REGION Network 5
   RUNG wire#powerrail
      "S2_Interlocks_DB"(Vessel_Rad_Level := "S2_General_Setup".Vessel_Rad_Level, Vessel_Rad_High_Alarm := "S2_General_Setup".Vessel_Alarm_Level, Pump_Rad_Level := "S2_General_Setup".Pump_Rad_Level, Pump_Rad_High_Alarm := "S2_General_Setup".Pump_Alarm_Level, Estop1 := "Estop1_PB_Active", Estop2 := "Estop2_PB_Active", Safety_Relay_Trip := "Safety_Relay_Trip", Safety_Lock_Engaged := "Safety_Lock2_Engaged", Manual_Mode := "S2_General_Setup".Manual_Mode, Rad_Lock_Bypass := "S2_General_Setup".Rad_Lock_Bypass, Process_Complete := "S2_General_Setup".Auto_Process_Complete, Water_Supply_Interlock := "S2_General_Setup".Water_Supply_Interlock, UM_Container_Interlock := "Setup_Data".Waste_Container_Interlock, UM_Container_HH_Interlock := "UM_HI_Level_SW", Buzzer_Reset := "Setup_Data".Buzzer_Reset, Rad_Lock := "S2_General_Setup".Rad_Lock, Estop_Active := "Setup_Data".Estop_Active, Level_Interlock := "S2_General_Setup".Level_Interlock, Pump_Permisive => "Pmp2_Permissive")
   END_RUNG
   // the same network as SCL:
   "S2_Interlocks_DB"(Vessel_Rad_Level := "S2_General_Setup".Vessel_Rad_Level,   // "Interlocks"
                      Vessel_Rad_High_Alarm := "S2_General_Setup".Vessel_Alarm_Level,
                      Pump_Rad_Level := "S2_General_Setup".Pump_Rad_Level,
                      Pump_Rad_High_Alarm := "S2_General_Setup".Pump_Alarm_Level,
                      Estop1 := "Estop1_PB_Active",
                      Estop2 := "Estop2_PB_Active",
                      Safety_Relay_Trip := "Safety_Relay_Trip",
                      Safety_Lock_Engaged := "Safety_Lock2_Engaged",
                      Manual_Mode := "S2_General_Setup".Manual_Mode,
                      Rad_Lock_Bypass := "S2_General_Setup".Rad_Lock_Bypass,
                      Process_Complete := "S2_General_Setup".Auto_Process_Complete,
                      Water_Supply_Interlock := "S2_General_Setup".Water_Supply_Interlock,
                      UM_Container_Interlock := "Setup_Data".Waste_Container_Interlock,
                      UM_Container_HH_Interlock := "UM_HI_Level_SW",
                      Buzzer_Reset := "Setup_Data".Buzzer_Reset,
                      Rad_Lock := "S2_General_Setup".Rad_Lock,
                      Estop_Active := "Setup_Data".Estop_Active,
                      Level_Interlock := "S2_General_Setup".Level_Interlock,
                      Pump_Permisive => "Pmp2_Permissive");
END_REGION

REGION Network 6
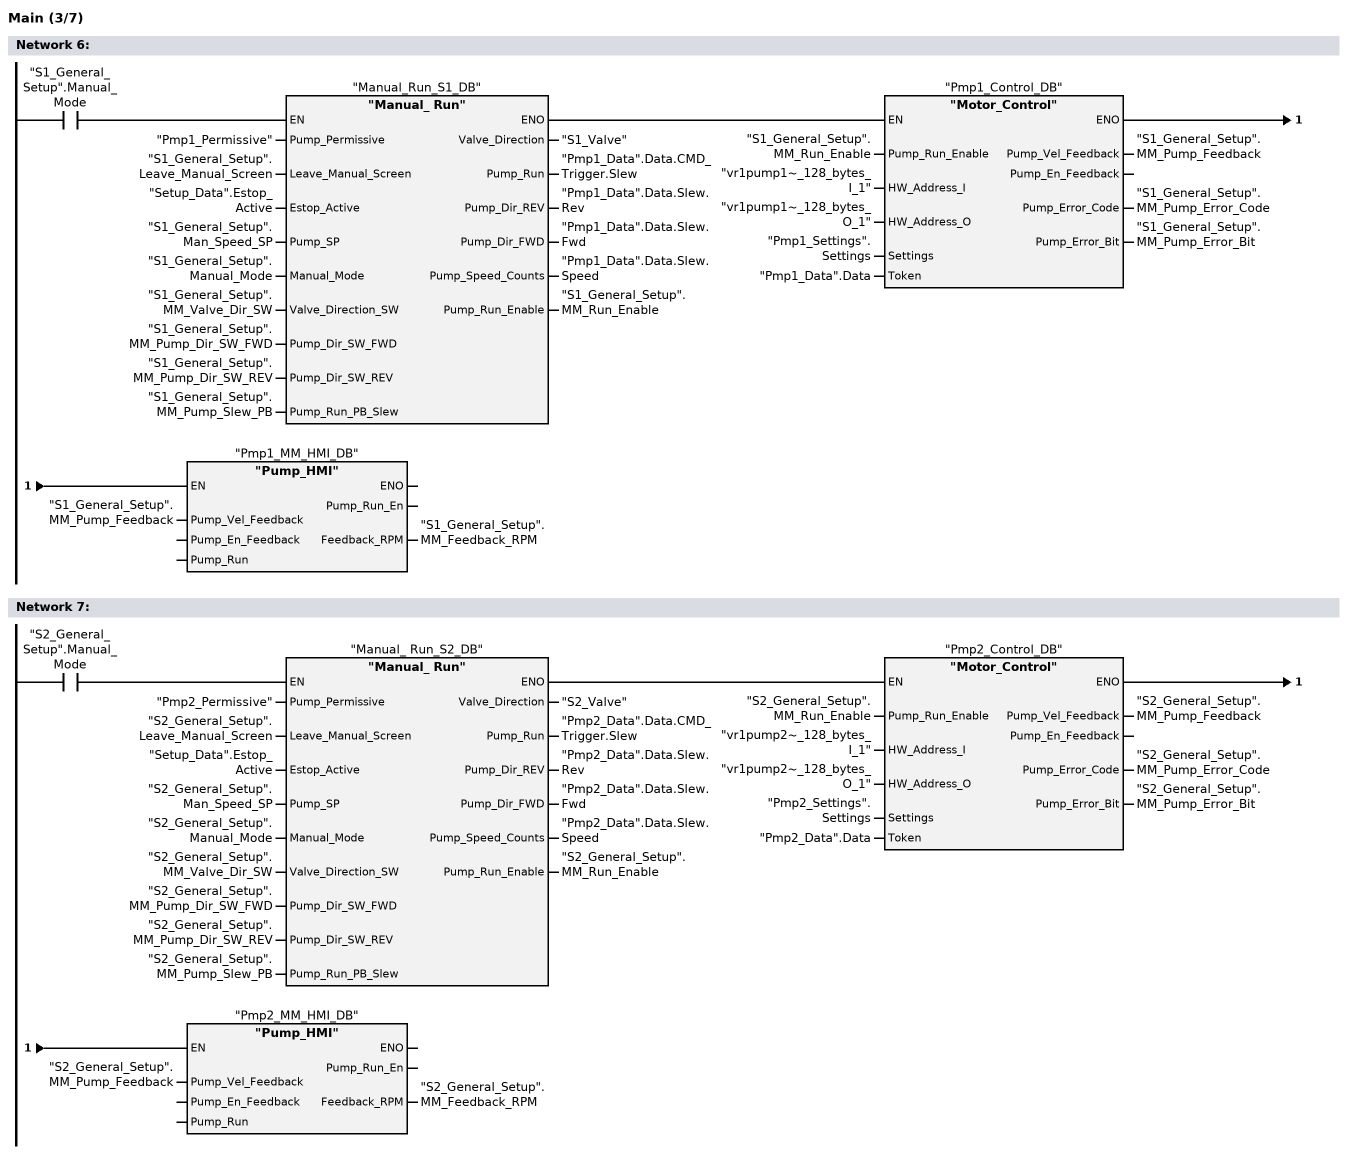
   RUNG wire#powerrail
      Contact( "S1_General_Setup".Manual_Mode )
      "Manual_Run_S1_DB"(Pump_Permissive := "Pmp1_Permissive", Leave_Manual_Screen := "S1_General_Setup".Leave_Manual_Screen, Estop_Active := "Setup_Data".Estop_Active, Pump_SP := "S1_General_Setup".Man_Speed_SP, Manual_Mode := "S1_General_Setup".Manual_Mode, Valve_Direction_SW := "S1_General_Setup".MM_Valve_Dir_SW, Pump_Dir_SW_FWD := "S1_General_Setup".MM_Pump_Dir_SW_FWD, Pump_Dir_SW_REV := "S1_General_Setup".MM_Pump_Dir_SW_REV, Pump_Run_PB_Slew := "S1_General_Setup".MM_Pump_Slew_PB, Valve_Direction => "S1_Valve", Pump_Run => "Pmp1_Data".Data.CMD_Trigger.Slew, Pump_Dir_REV => "Pmp1_Data".Data.Slew.Rev, Pump_Dir_FWD => "Pmp1_Data".Data.Slew.Fwd, Pump_Speed_Counts => "Pmp1_Data".Data.Slew.Speed, Pump_Run_Enable => "S1_General_Setup".MM_Run_Enable)
      "Pmp1_Control_DB"(Pump_Run_Enable := "S1_General_Setup".MM_Run_Enable, HW_Address_I := "vr1pump1~_128_bytes_I_1", HW_Address_O := "vr1pump1~_128_bytes_O_1", Settings := "Pmp1_Settings".Settings, Token := "Pmp1_Data".Data, Pump_Vel_Feedback => "S1_General_Setup".MM_Pump_Feedback, Pump_En_Feedback =>, Pump_Error_Code => "S1_General_Setup".MM_Pump_Error_Code, Pump_Error_Bit => "S1_General_Setup".MM_Pump_Error_Bit)
      "Pmp1_MM_HMI_DB"(Pump_Vel_Feedback := "S1_General_Setup".MM_Pump_Feedback, Pump_En_Feedback :=, Pump_Run :=, Pump_Run_En =>, Feedback_RPM => "S1_General_Setup".MM_Feedback_RPM)
   END_RUNG
   // the same network as SCL:
   "Manual_Run_S1_DB"(EN := "S1_General_Setup".Manual_Mode,   // "Manual_ Run"
                      Pump_Permissive := "Pmp1_Permissive",
                      Leave_Manual_Screen := "S1_General_Setup".Leave_Manual_Screen,
                      Estop_Active := "Setup_Data".Estop_Active,
                      Pump_SP := "S1_General_Setup".Man_Speed_SP,
                      Manual_Mode := "S1_General_Setup".Manual_Mode,
                      Valve_Direction_SW := "S1_General_Setup".MM_Valve_Dir_SW,
                      Pump_Dir_SW_FWD := "S1_General_Setup".MM_Pump_Dir_SW_FWD,
                      Pump_Dir_SW_REV := "S1_General_Setup".MM_Pump_Dir_SW_REV,
                      Pump_Run_PB_Slew := "S1_General_Setup".MM_Pump_Slew_PB,
                      Valve_Direction => "S1_Valve",
                      Pump_Run => "Pmp1_Data".Data.CMD_Trigger.Slew,
                      Pump_Dir_REV => "Pmp1_Data".Data.Slew.Rev,
                      Pump_Dir_FWD => "Pmp1_Data".Data.Slew.Fwd,
                      Pump_Speed_Counts => "Pmp1_Data".Data.Slew.Speed,
                      Pump_Run_Enable => "S1_General_Setup".MM_Run_Enable,
                      ENO => #_w1);
   "Pmp1_Control_DB"(EN := #_w1,   // "Motor_Control"
                     Pump_Run_Enable := "S1_General_Setup".MM_Run_Enable,
                     HW_Address_I := "vr1pump1~_128_bytes_I_1",
                     HW_Address_O := "vr1pump1~_128_bytes_O_1",
                     Settings := "Pmp1_Settings".Settings,
                     Token := "Pmp1_Data".Data,
                     Pump_Vel_Feedback => "S1_General_Setup".MM_Pump_Feedback,
                     Pump_Error_Code => "S1_General_Setup".MM_Pump_Error_Code,
                     Pump_Error_Bit => "S1_General_Setup".MM_Pump_Error_Bit,
                     ENO => #_w2);
   IF #_w2 THEN
       "Pmp1_MM_HMI_DB"(Pump_Vel_Feedback := "S1_General_Setup".MM_Pump_Feedback,   // "Pump_HMI"
                        Feedback_RPM => "S1_General_Setup".MM_Feedback_RPM);
   END_IF;
END_REGION

REGION Network 7
   RUNG wire#powerrail
      Contact( "S2_General_Setup".Manual_Mode )
      "Manual_ Run_S2_DB"(Pump_Permissive := "Pmp2_Permissive", Leave_Manual_Screen := "S2_General_Setup".Leave_Manual_Screen, Estop_Active := "Setup_Data".Estop_Active, Pump_SP := "S2_General_Setup".Man_Speed_SP, Manual_Mode := "S2_General_Setup".Manual_Mode, Valve_Direction_SW := "S2_General_Setup".MM_Valve_Dir_SW, Pump_Dir_SW_FWD := "S2_General_Setup".MM_Pump_Dir_SW_FWD, Pump_Dir_SW_REV := "S2_General_Setup".MM_Pump_Dir_SW_REV, Pump_Run_PB_Slew := "S2_General_Setup".MM_Pump_Slew_PB, Valve_Direction => "S2_Valve", Pump_Run => "Pmp2_Data".Data.CMD_Trigger.Slew, Pump_Dir_REV => "Pmp2_Data".Data.Slew.Rev, Pump_Dir_FWD => "Pmp2_Data".Data.Slew.Fwd, Pump_Speed_Counts => "Pmp2_Data".Data.Slew.Speed, Pump_Run_Enable => "S2_General_Setup".MM_Run_Enable)
      "Pmp2_Control_DB"(Pump_Run_Enable := "S2_General_Setup".MM_Run_Enable, HW_Address_I := "vr1pump2~_128_bytes_I_1", HW_Address_O := "vr1pump2~_128_bytes_O_1", Settings := "Pmp2_Settings".Settings, Token := "Pmp2_Data".Data, Pump_Vel_Feedback => "S2_General_Setup".MM_Pump_Feedback, Pump_En_Feedback =>, Pump_Error_Code => "S2_General_Setup".MM_Pump_Error_Code, Pump_Error_Bit => "S2_General_Setup".MM_Pump_Error_Bit)
      "Pmp2_MM_HMI_DB"(Pump_Vel_Feedback := "S2_General_Setup".MM_Pump_Feedback, Pump_En_Feedback :=, Pump_Run :=, Pump_Run_En =>, Feedback_RPM => "S2_General_Setup".MM_Feedback_RPM)
   END_RUNG
   // the same network as SCL:
   "Manual_ Run_S2_DB"(EN := "S2_General_Setup".Manual_Mode,   // "Manual_ Run"
                       Pump_Permissive := "Pmp2_Permissive",
                       Leave_Manual_Screen := "S2_General_Setup".Leave_Manual_Screen,
                       Estop_Active := "Setup_Data".Estop_Active,
                       Pump_SP := "S2_General_Setup".Man_Speed_SP,
                       Manual_Mode := "S2_General_Setup".Manual_Mode,
                       Valve_Direction_SW := "S2_General_Setup".MM_Valve_Dir_SW,
                       Pump_Dir_SW_FWD := "S2_General_Setup".MM_Pump_Dir_SW_FWD,
                       Pump_Dir_SW_REV := "S2_General_Setup".MM_Pump_Dir_SW_REV,
                       Pump_Run_PB_Slew := "S2_General_Setup".MM_Pump_Slew_PB,
                       Valve_Direction => "S2_Valve",
                       Pump_Run => "Pmp2_Data".Data.CMD_Trigger.Slew,
                       Pump_Dir_REV => "Pmp2_Data".Data.Slew.Rev,
                       Pump_Dir_FWD => "Pmp2_Data".Data.Slew.Fwd,
                       Pump_Speed_Counts => "Pmp2_Data".Data.Slew.Speed,
                       Pump_Run_Enable => "S2_General_Setup".MM_Run_Enable,
                       ENO => #_w1);
   "Pmp2_Control_DB"(EN := #_w1,   // "Motor_Control"
                     Pump_Run_Enable := "S2_General_Setup".MM_Run_Enable,
                     HW_Address_I := "vr1pump2~_128_bytes_I_1",
                     HW_Address_O := "vr1pump2~_128_bytes_O_1",
                     Settings := "Pmp2_Settings".Settings,
                     Token := "Pmp2_Data".Data,
                     Pump_Vel_Feedback => "S2_General_Setup".MM_Pump_Feedback,
                     Pump_Error_Code => "S2_General_Setup".MM_Pump_Error_Code,
                     Pump_Error_Bit => "S2_General_Setup".MM_Pump_Error_Bit,
                     ENO => #_w2);
   IF #_w2 THEN
       "Pmp2_MM_HMI_DB"(Pump_Vel_Feedback := "S2_General_Setup".MM_Pump_Feedback,   // "Pump_HMI"
                        Feedback_RPM => "S2_General_Setup".MM_Feedback_RPM);
   END_IF;
END_REGION

REGION Network 8
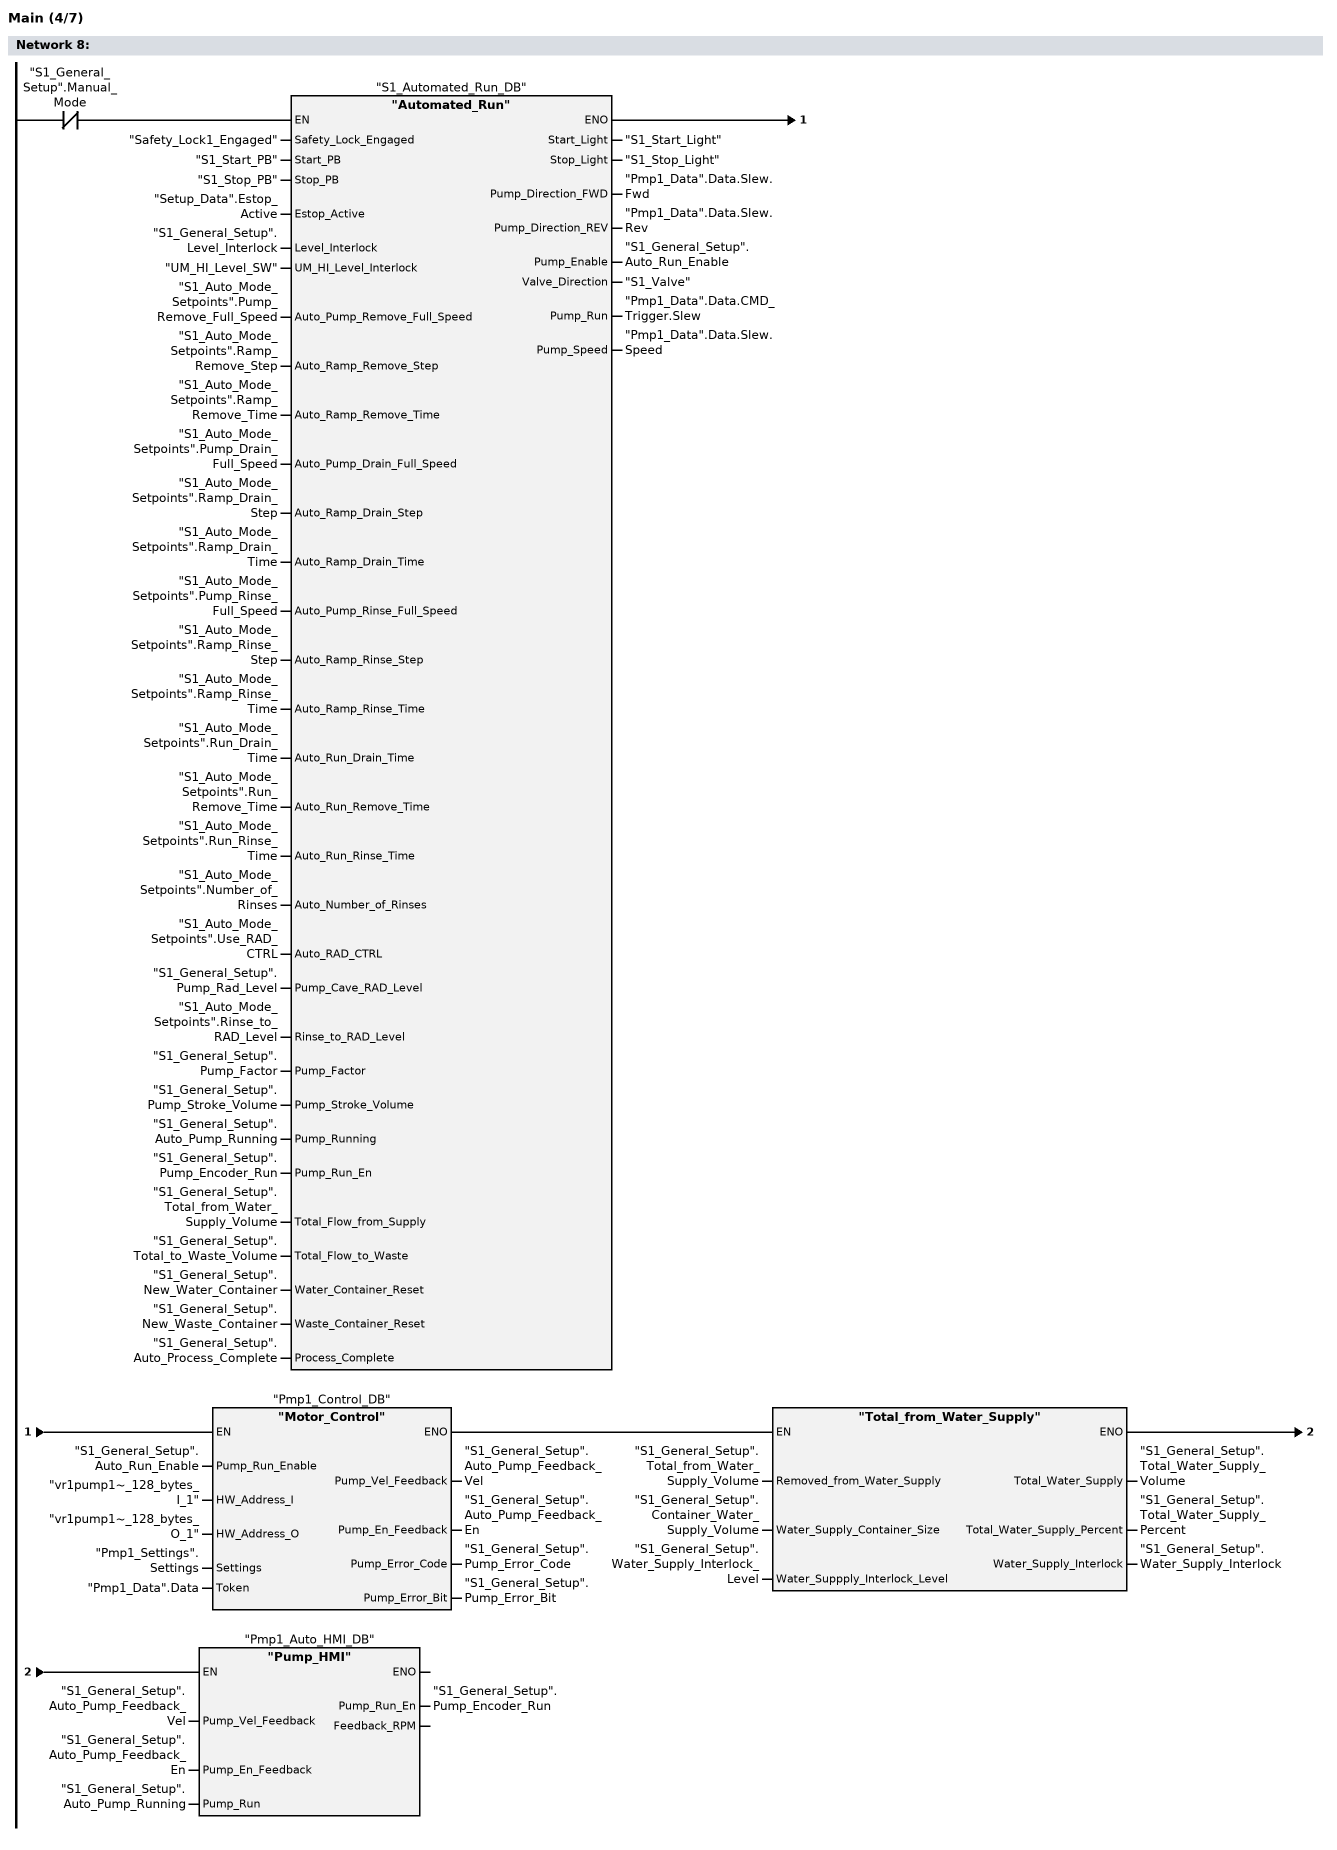
   RUNG wire#powerrail
      I_Contact( "S1_General_Setup".Manual_Mode )
      "S1_Automated_Run_DB"(Safety_Lock_Engaged := "Safety_Lock1_Engaged", Start_PB := "S1_Start_PB", Stop_PB := "S1_Stop_PB", Estop_Active := "Setup_Data".Estop_Active, Level_Interlock := "S1_General_Setup".Level_Interlock, UM_HI_Level_Interlock := "UM_HI_Level_SW", Auto_Pump_Remove_Full_Speed := "S1_Auto_Mode_Setpoints".Pump_Remove_Full_Speed, Auto_Ramp_Remove_Step := "S1_Auto_Mode_Setpoints".Ramp_Remove_Step, Auto_Ramp_Remove_Time := "S1_Auto_Mode_Setpoints".Ramp_Remove_Time, Auto_Pump_Drain_Full_Speed := "S1_Auto_Mode_Setpoints".Pump_Drain_Full_Speed, Auto_Ramp_Drain_Step := "S1_Auto_Mode_Setpoints".Ramp_Drain_Step, Auto_Ramp_Drain_Time := "S1_Auto_Mode_Setpoints".Ramp_Drain_Time, Auto_Pump_Rinse_Full_Speed := "S1_Auto_Mode_Setpoints".Pump_Rinse_Full_Speed, Auto_Ramp_Rinse_Step := "S1_Auto_Mode_Setpoints".Ramp_Rinse_Step, Auto_Ramp_Rinse_Time := "S1_Auto_Mode_Setpoints".Ramp_Rinse_Time, Auto_Run_Drain_Time := "S1_Auto_Mode_Setpoints".Run_Drain_Time, Auto_Run_Remove_Time := "S1_Auto_Mode_Setpoints".Run_Remove_Time, Auto_Run_Rinse_Time := "S1_Auto_Mode_Setpoints".Run_Rinse_Time, Auto_Number_of_Rinses := "S1_Auto_Mode_Setpoints".Number_of_Rinses, Auto_RAD_CTRL := "S1_Auto_Mode_Setpoints".Use_RAD_CTRL, Pump_Cave_RAD_Level := "S1_General_Setup".Pump_Rad_Level, Rinse_to_RAD_Level := "S1_Auto_Mode_Setpoints".Rinse_to_RAD_Level, Pump_Factor := "S1_General_Setup".Pump_Factor, Pump_Stroke_Volume := "S1_General_Setup".Pump_Stroke_Volume, Pump_Running := "S1_General_Setup".Auto_Pump_Running, Pump_Run_En := "S1_General_Setup".Pump_Encoder_Run, Total_Flow_from_Supply := "S1_General_Setup".Total_from_Water_Supply_Volume, Total_Flow_to_Waste := "S1_General_Setup".Total_to_Waste_Volume, Water_Container_Reset := "S1_General_Setup".New_Water_Container, Waste_Container_Reset := "S1_General_Setup".New_Waste_Container, Process_Complete := "S1_General_Setup".Auto_Process_Complete, Start_Light => "S1_Start_Light", Stop_Light => "S1_Stop_Light", Pump_Direction_FWD => "Pmp1_Data".Data.Slew.Fwd, Pump_Direction_REV => "Pmp1_Data".Data.Slew.Rev, Pump_Enable => "S1_General_Setup".Auto_Run_Enable, Valve_Direction => "S1_Valve", Pump_Run => "Pmp1_Data".Data.CMD_Trigger.Slew, Pump_Speed => "Pmp1_Data".Data.Slew.Speed)
      "Pmp1_Control_DB"(Pump_Run_Enable := "S1_General_Setup".Auto_Run_Enable, HW_Address_I := "vr1pump1~_128_bytes_I_1", HW_Address_O := "vr1pump1~_128_bytes_O_1", Settings := "Pmp1_Settings".Settings, Token := "Pmp1_Data".Data, Pump_Vel_Feedback => "S1_General_Setup".Auto_Pump_Feedback_Vel, Pump_En_Feedback => "S1_General_Setup".Auto_Pump_Feedback_En, Pump_Error_Code => "S1_General_Setup".Pump_Error_Code, Pump_Error_Bit => "S1_General_Setup".Pump_Error_Bit)
      "Total_from_Water_Supply"(Removed_from_Water_Supply := "S1_General_Setup".Total_from_Water_Supply_Volume, Water_Supply_Container_Size := "S1_General_Setup".Container_Water_Supply_Volume, Water_Suppply_Interlock_Level := "S1_General_Setup".Water_Supply_Interlock_Level, Total_Water_Supply => "S1_General_Setup".Total_Water_Supply_Volume, Total_Water_Supply_Percent => "S1_General_Setup".Total_Water_Supply_Percent, Water_Supply_Interlock => "S1_General_Setup".Water_Supply_Interlock)
      "Pmp1_Auto_HMI_DB"(Pump_Vel_Feedback := "S1_General_Setup".Auto_Pump_Feedback_Vel, Pump_En_Feedback := "S1_General_Setup".Auto_Pump_Feedback_En, Pump_Run := "S1_General_Setup".Auto_Pump_Running, Pump_Run_En => "S1_General_Setup".Pump_Encoder_Run, Feedback_RPM =>)
   END_RUNG
   // the same network as SCL:
   "S1_Automated_Run_DB"(EN := NOT "S1_General_Setup".Manual_Mode,   // "Automated_Run"
                         Safety_Lock_Engaged := "Safety_Lock1_Engaged",
                         Start_PB := "S1_Start_PB",
                         Stop_PB := "S1_Stop_PB",
                         Estop_Active := "Setup_Data".Estop_Active,
                         Level_Interlock := "S1_General_Setup".Level_Interlock,
                         UM_HI_Level_Interlock := "UM_HI_Level_SW",
                         Auto_Pump_Remove_Full_Speed := "S1_Auto_Mode_Setpoints".Pump_Remove_Full_Speed,
                         Auto_Ramp_Remove_Step := "S1_Auto_Mode_Setpoints".Ramp_Remove_Step,
                         Auto_Ramp_Remove_Time := "S1_Auto_Mode_Setpoints".Ramp_Remove_Time,
                         Auto_Pump_Drain_Full_Speed := "S1_Auto_Mode_Setpoints".Pump_Drain_Full_Speed,
                         Auto_Ramp_Drain_Step := "S1_Auto_Mode_Setpoints".Ramp_Drain_Step,
                         Auto_Ramp_Drain_Time := "S1_Auto_Mode_Setpoints".Ramp_Drain_Time,
                         Auto_Pump_Rinse_Full_Speed := "S1_Auto_Mode_Setpoints".Pump_Rinse_Full_Speed,
                         Auto_Ramp_Rinse_Step := "S1_Auto_Mode_Setpoints".Ramp_Rinse_Step,
                         Auto_Ramp_Rinse_Time := "S1_Auto_Mode_Setpoints".Ramp_Rinse_Time,
                         Auto_Run_Drain_Time := "S1_Auto_Mode_Setpoints".Run_Drain_Time,
                         Auto_Run_Remove_Time := "S1_Auto_Mode_Setpoints".Run_Remove_Time,
                         Auto_Run_Rinse_Time := "S1_Auto_Mode_Setpoints".Run_Rinse_Time,
                         Auto_Number_of_Rinses := "S1_Auto_Mode_Setpoints".Number_of_Rinses,
                         Auto_RAD_CTRL := "S1_Auto_Mode_Setpoints".Use_RAD_CTRL,
                         Pump_Cave_RAD_Level := "S1_General_Setup".Pump_Rad_Level,
                         Rinse_to_RAD_Level := "S1_Auto_Mode_Setpoints".Rinse_to_RAD_Level,
                         Pump_Factor := "S1_General_Setup".Pump_Factor,
                         Pump_Stroke_Volume := "S1_General_Setup".Pump_Stroke_Volume,
                         Pump_Running := "S1_General_Setup".Auto_Pump_Running,
                         Pump_Run_En := "S1_General_Setup".Pump_Encoder_Run,
                         Total_Flow_from_Supply := "S1_General_Setup".Total_from_Water_Supply_Volume,
                         Total_Flow_to_Waste := "S1_General_Setup".Total_to_Waste_Volume,
                         Water_Container_Reset := "S1_General_Setup".New_Water_Container,
                         Waste_Container_Reset := "S1_General_Setup".New_Waste_Container,
                         Process_Complete := "S1_General_Setup".Auto_Process_Complete,
                         Start_Light => "S1_Start_Light",
                         Stop_Light => "S1_Stop_Light",
                         Pump_Direction_FWD => "Pmp1_Data".Data.Slew.Fwd,
                         Pump_Direction_REV => "Pmp1_Data".Data.Slew.Rev,
                         Pump_Enable => "S1_General_Setup".Auto_Run_Enable,
                         Valve_Direction => "S1_Valve",
                         Pump_Run => "Pmp1_Data".Data.CMD_Trigger.Slew,
                         Pump_Speed => "Pmp1_Data".Data.Slew.Speed,
                         ENO => #_w1);
   "Pmp1_Control_DB"(EN := #_w1,   // "Motor_Control"
                     Pump_Run_Enable := "S1_General_Setup".Auto_Run_Enable,
                     HW_Address_I := "vr1pump1~_128_bytes_I_1",
                     HW_Address_O := "vr1pump1~_128_bytes_O_1",
                     Settings := "Pmp1_Settings".Settings,
                     Token := "Pmp1_Data".Data,
                     Pump_Vel_Feedback => "S1_General_Setup".Auto_Pump_Feedback_Vel,
                     Pump_En_Feedback => "S1_General_Setup".Auto_Pump_Feedback_En,
                     Pump_Error_Code => "S1_General_Setup".Pump_Error_Code,
                     Pump_Error_Bit => "S1_General_Setup".Pump_Error_Bit,
                     ENO => #_w2);
   "Total_from_Water_Supply"(EN := #_w2,
                           Removed_from_Water_Supply := "S1_General_Setup".Total_from_Water_Supply_Volume,
                           Water_Supply_Container_Size := "S1_General_Setup".Container_Water_Supply_Volume,
                           Water_Suppply_Interlock_Level := "S1_General_Setup".Water_Supply_Interlock_Level,
                           Total_Water_Supply => "S1_General_Setup".Total_Water_Supply_Volume,
                           Total_Water_Supply_Percent => "S1_General_Setup".Total_Water_Supply_Percent,
                           Water_Supply_Interlock => "S1_General_Setup".Water_Supply_Interlock,
                           ENO => #_w3);
   IF #_w3 THEN
       "Pmp1_Auto_HMI_DB"(Pump_Vel_Feedback := "S1_General_Setup".Auto_Pump_Feedback_Vel,   // "Pump_HMI"
                          Pump_En_Feedback := "S1_General_Setup".Auto_Pump_Feedback_En,
                          Pump_Run := "S1_General_Setup".Auto_Pump_Running,
                          Pump_Run_En => "S1_General_Setup".Pump_Encoder_Run);
   END_IF;
END_REGION

REGION Network 9
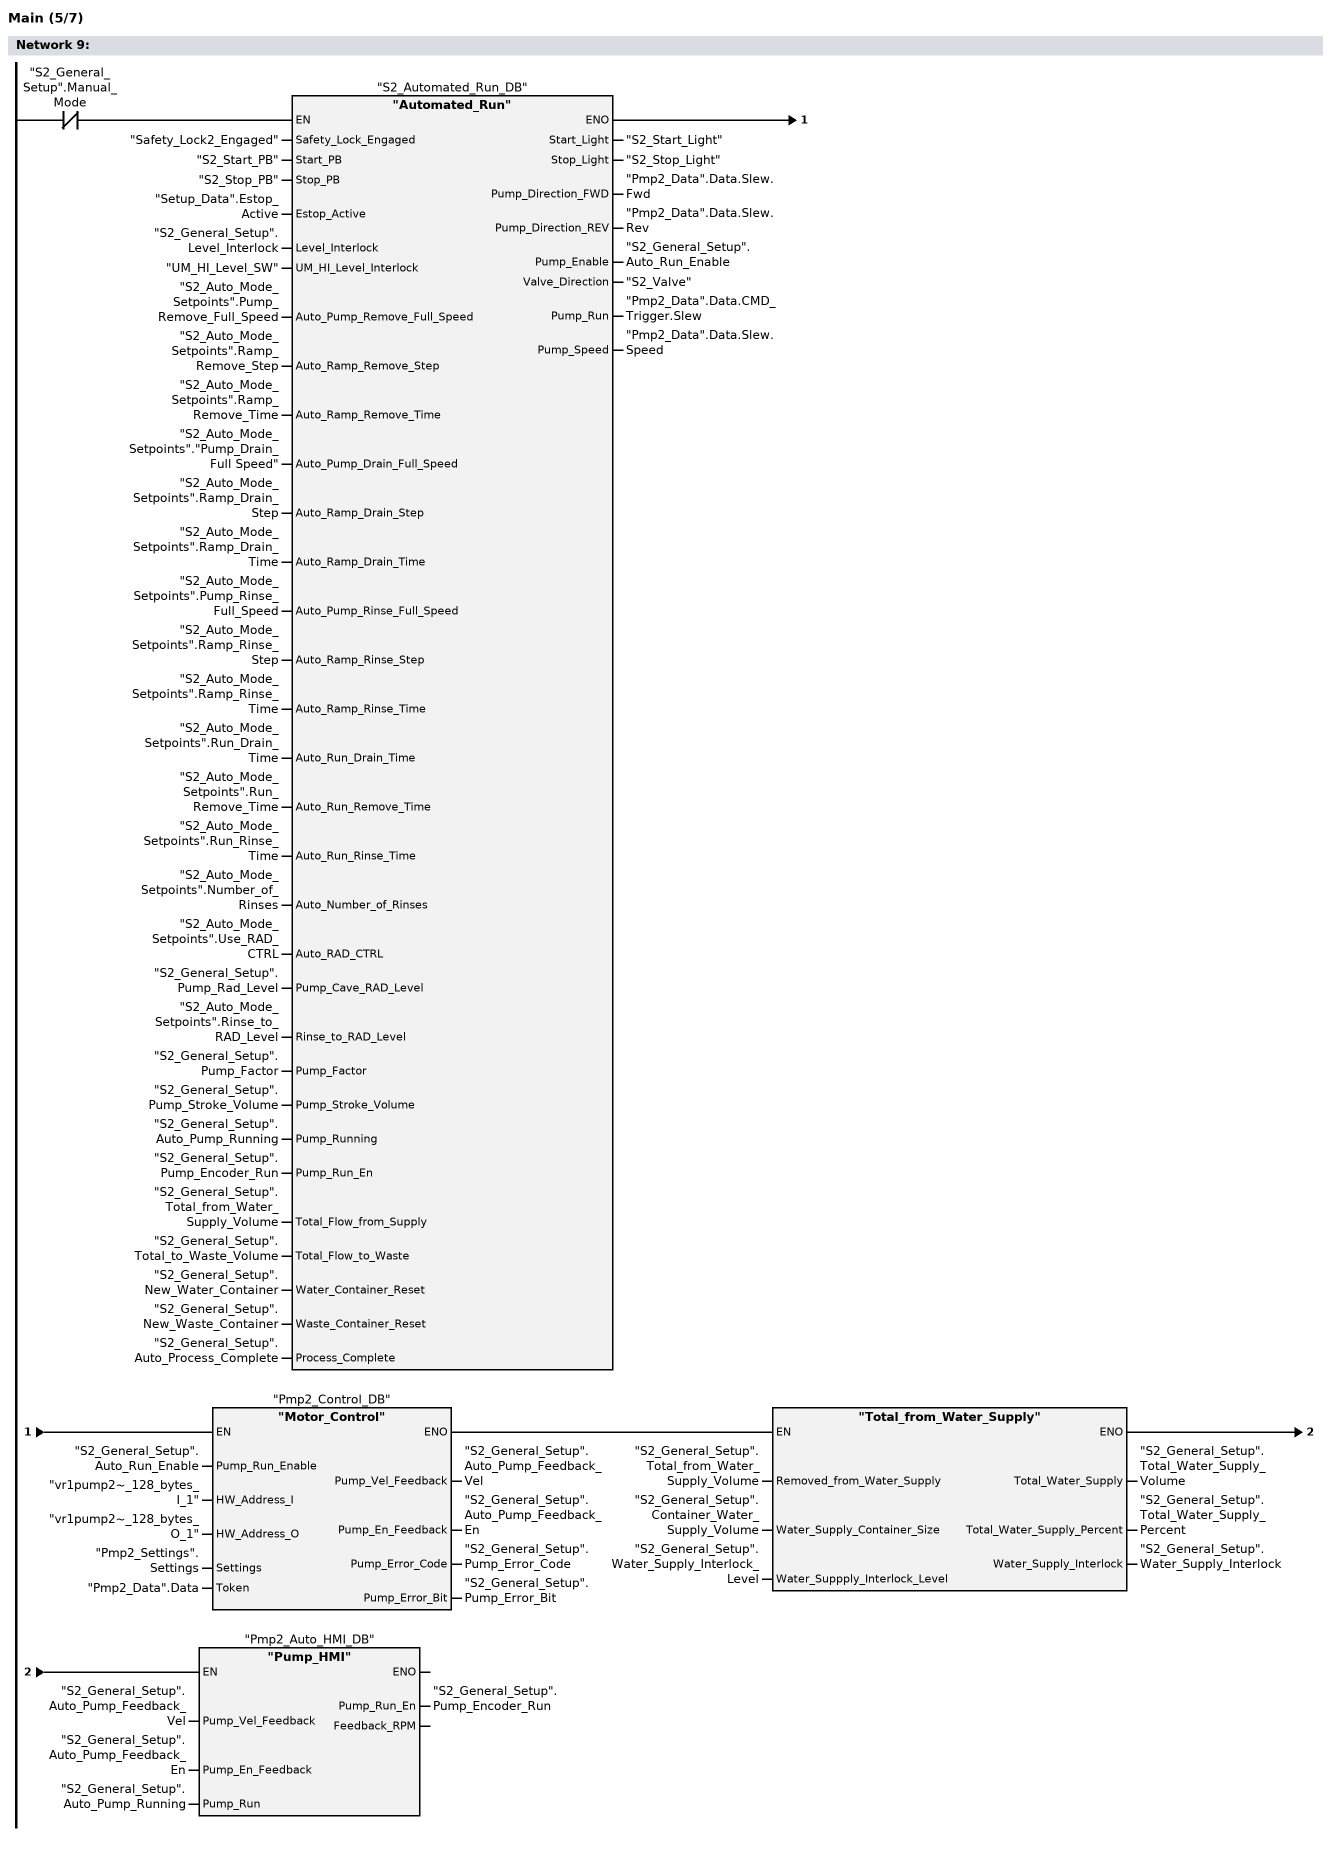
   RUNG wire#powerrail
      I_Contact( "S2_General_Setup".Manual_Mode )
      "S2_Automated_Run_DB"(Safety_Lock_Engaged := "Safety_Lock2_Engaged", Start_PB := "S2_Start_PB", Stop_PB := "S2_Stop_PB", Estop_Active := "Setup_Data".Estop_Active, Level_Interlock := "S2_General_Setup".Level_Interlock, UM_HI_Level_Interlock := "UM_HI_Level_SW", Auto_Pump_Remove_Full_Speed := "S2_Auto_Mode_Setpoints".Pump_Remove_Full_Speed, Auto_Ramp_Remove_Step := "S2_Auto_Mode_Setpoints".Ramp_Remove_Step, Auto_Ramp_Remove_Time := "S2_Auto_Mode_Setpoints".Ramp_Remove_Time, Auto_Pump_Drain_Full_Speed := "S2_Auto_Mode_Setpoints"."Pump_Drain_Full Speed", Auto_Ramp_Drain_Step := "S2_Auto_Mode_Setpoints".Ramp_Drain_Step, Auto_Ramp_Drain_Time := "S2_Auto_Mode_Setpoints".Ramp_Drain_Time, Auto_Pump_Rinse_Full_Speed := "S2_Auto_Mode_Setpoints".Pump_Rinse_Full_Speed, Auto_Ramp_Rinse_Step := "S2_Auto_Mode_Setpoints".Ramp_Rinse_Step, Auto_Ramp_Rinse_Time := "S2_Auto_Mode_Setpoints".Ramp_Rinse_Time, Auto_Run_Drain_Time := "S2_Auto_Mode_Setpoints".Run_Drain_Time, Auto_Run_Remove_Time := "S2_Auto_Mode_Setpoints".Run_Remove_Time, Auto_Run_Rinse_Time := "S2_Auto_Mode_Setpoints".Run_Rinse_Time, Auto_Number_of_Rinses := "S2_Auto_Mode_Setpoints".Number_of_Rinses, Auto_RAD_CTRL := "S2_Auto_Mode_Setpoints".Use_RAD_CTRL, Pump_Cave_RAD_Level := "S2_General_Setup".Pump_Rad_Level, Rinse_to_RAD_Level := "S2_Auto_Mode_Setpoints".Rinse_to_RAD_Level, Pump_Factor := "S2_General_Setup".Pump_Factor, Pump_Stroke_Volume := "S2_General_Setup".Pump_Stroke_Volume, Pump_Running := "S2_General_Setup".Auto_Pump_Running, Pump_Run_En := "S2_General_Setup".Pump_Encoder_Run, Total_Flow_from_Supply := "S2_General_Setup".Total_from_Water_Supply_Volume, Total_Flow_to_Waste := "S2_General_Setup".Total_to_Waste_Volume, Water_Container_Reset := "S2_General_Setup".New_Water_Container, Waste_Container_Reset := "S2_General_Setup".New_Waste_Container, Process_Complete := "S2_General_Setup".Auto_Process_Complete, Start_Light => "S2_Start_Light", Stop_Light => "S2_Stop_Light", Pump_Direction_FWD => "Pmp2_Data".Data.Slew.Fwd, Pump_Direction_REV => "Pmp2_Data".Data.Slew.Rev, Pump_Enable => "S2_General_Setup".Auto_Run_Enable, Valve_Direction => "S2_Valve", Pump_Run => "Pmp2_Data".Data.CMD_Trigger.Slew, Pump_Speed => "Pmp2_Data".Data.Slew.Speed)
      "Pmp2_Control_DB"(Pump_Run_Enable := "S2_General_Setup".Auto_Run_Enable, HW_Address_I := "vr1pump2~_128_bytes_I_1", HW_Address_O := "vr1pump2~_128_bytes_O_1", Settings := "Pmp2_Settings".Settings, Token := "Pmp2_Data".Data, Pump_Vel_Feedback => "S2_General_Setup".Auto_Pump_Feedback_Vel, Pump_En_Feedback => "S2_General_Setup".Auto_Pump_Feedback_En, Pump_Error_Code => "S2_General_Setup".Pump_Error_Code, Pump_Error_Bit => "S2_General_Setup".Pump_Error_Bit)
      "Total_from_Water_Supply"(Removed_from_Water_Supply := "S2_General_Setup".Total_from_Water_Supply_Volume, Water_Supply_Container_Size := "S2_General_Setup".Container_Water_Supply_Volume, Water_Suppply_Interlock_Level := "S2_General_Setup".Water_Supply_Interlock_Level, Total_Water_Supply => "S2_General_Setup".Total_Water_Supply_Volume, Total_Water_Supply_Percent => "S2_General_Setup".Total_Water_Supply_Percent, Water_Supply_Interlock => "S2_General_Setup".Water_Supply_Interlock)
      "Pmp2_Auto_HMI_DB"(Pump_Vel_Feedback := "S2_General_Setup".Auto_Pump_Feedback_Vel, Pump_En_Feedback := "S2_General_Setup".Auto_Pump_Feedback_En, Pump_Run := "S2_General_Setup".Auto_Pump_Running, Pump_Run_En => "S2_General_Setup".Pump_Encoder_Run, Feedback_RPM =>)
   END_RUNG
   // the same network as SCL:
   "S2_Automated_Run_DB"(EN := NOT "S2_General_Setup".Manual_Mode,   // "Automated_Run"
                         Safety_Lock_Engaged := "Safety_Lock2_Engaged",
                         Start_PB := "S2_Start_PB",
                         Stop_PB := "S2_Stop_PB",
                         Estop_Active := "Setup_Data".Estop_Active,
                         Level_Interlock := "S2_General_Setup".Level_Interlock,
                         UM_HI_Level_Interlock := "UM_HI_Level_SW",
                         Auto_Pump_Remove_Full_Speed := "S2_Auto_Mode_Setpoints".Pump_Remove_Full_Speed,
                         Auto_Ramp_Remove_Step := "S2_Auto_Mode_Setpoints".Ramp_Remove_Step,
                         Auto_Ramp_Remove_Time := "S2_Auto_Mode_Setpoints".Ramp_Remove_Time,
                         Auto_Pump_Drain_Full_Speed := "S2_Auto_Mode_Setpoints"."Pump_Drain_Full Speed",
                         Auto_Ramp_Drain_Step := "S2_Auto_Mode_Setpoints".Ramp_Drain_Step,
                         Auto_Ramp_Drain_Time := "S2_Auto_Mode_Setpoints".Ramp_Drain_Time,
                         Auto_Pump_Rinse_Full_Speed := "S2_Auto_Mode_Setpoints".Pump_Rinse_Full_Speed,
                         Auto_Ramp_Rinse_Step := "S2_Auto_Mode_Setpoints".Ramp_Rinse_Step,
                         Auto_Ramp_Rinse_Time := "S2_Auto_Mode_Setpoints".Ramp_Rinse_Time,
                         Auto_Run_Drain_Time := "S2_Auto_Mode_Setpoints".Run_Drain_Time,
                         Auto_Run_Remove_Time := "S2_Auto_Mode_Setpoints".Run_Remove_Time,
                         Auto_Run_Rinse_Time := "S2_Auto_Mode_Setpoints".Run_Rinse_Time,
                         Auto_Number_of_Rinses := "S2_Auto_Mode_Setpoints".Number_of_Rinses,
                         Auto_RAD_CTRL := "S2_Auto_Mode_Setpoints".Use_RAD_CTRL,
                         Pump_Cave_RAD_Level := "S2_General_Setup".Pump_Rad_Level,
                         Rinse_to_RAD_Level := "S2_Auto_Mode_Setpoints".Rinse_to_RAD_Level,
                         Pump_Factor := "S2_General_Setup".Pump_Factor,
                         Pump_Stroke_Volume := "S2_General_Setup".Pump_Stroke_Volume,
                         Pump_Running := "S2_General_Setup".Auto_Pump_Running,
                         Pump_Run_En := "S2_General_Setup".Pump_Encoder_Run,
                         Total_Flow_from_Supply := "S2_General_Setup".Total_from_Water_Supply_Volume,
                         Total_Flow_to_Waste := "S2_General_Setup".Total_to_Waste_Volume,
                         Water_Container_Reset := "S2_General_Setup".New_Water_Container,
                         Waste_Container_Reset := "S2_General_Setup".New_Waste_Container,
                         Process_Complete := "S2_General_Setup".Auto_Process_Complete,
                         Start_Light => "S2_Start_Light",
                         Stop_Light => "S2_Stop_Light",
                         Pump_Direction_FWD => "Pmp2_Data".Data.Slew.Fwd,
                         Pump_Direction_REV => "Pmp2_Data".Data.Slew.Rev,
                         Pump_Enable => "S2_General_Setup".Auto_Run_Enable,
                         Valve_Direction => "S2_Valve",
                         Pump_Run => "Pmp2_Data".Data.CMD_Trigger.Slew,
                         Pump_Speed => "Pmp2_Data".Data.Slew.Speed,
                         ENO => #_w1);
   "Pmp2_Control_DB"(EN := #_w1,   // "Motor_Control"
                     Pump_Run_Enable := "S2_General_Setup".Auto_Run_Enable,
                     HW_Address_I := "vr1pump2~_128_bytes_I_1",
                     HW_Address_O := "vr1pump2~_128_bytes_O_1",
                     Settings := "Pmp2_Settings".Settings,
                     Token := "Pmp2_Data".Data,
                     Pump_Vel_Feedback => "S2_General_Setup".Auto_Pump_Feedback_Vel,
                     Pump_En_Feedback => "S2_General_Setup".Auto_Pump_Feedback_En,
                     Pump_Error_Code => "S2_General_Setup".Pump_Error_Code,
                     Pump_Error_Bit => "S2_General_Setup".Pump_Error_Bit,
                     ENO => #_w2);
   "Total_from_Water_Supply"(EN := #_w2,
                           Removed_from_Water_Supply := "S2_General_Setup".Total_from_Water_Supply_Volume,
                           Water_Supply_Container_Size := "S2_General_Setup".Container_Water_Supply_Volume,
                           Water_Suppply_Interlock_Level := "S2_General_Setup".Water_Supply_Interlock_Level,
                           Total_Water_Supply => "S2_General_Setup".Total_Water_Supply_Volume,
                           Total_Water_Supply_Percent => "S2_General_Setup".Total_Water_Supply_Percent,
                           Water_Supply_Interlock => "S2_General_Setup".Water_Supply_Interlock,
                           ENO => #_w3);
   IF #_w3 THEN
       "Pmp2_Auto_HMI_DB"(Pump_Vel_Feedback := "S2_General_Setup".Auto_Pump_Feedback_Vel,   // "Pump_HMI"
                          Pump_En_Feedback := "S2_General_Setup".Auto_Pump_Feedback_En,
                          Pump_Run := "S2_General_Setup".Auto_Pump_Running,
                          Pump_Run_En => "S2_General_Setup".Pump_Encoder_Run);
   END_IF;
END_REGION

REGION Network 10
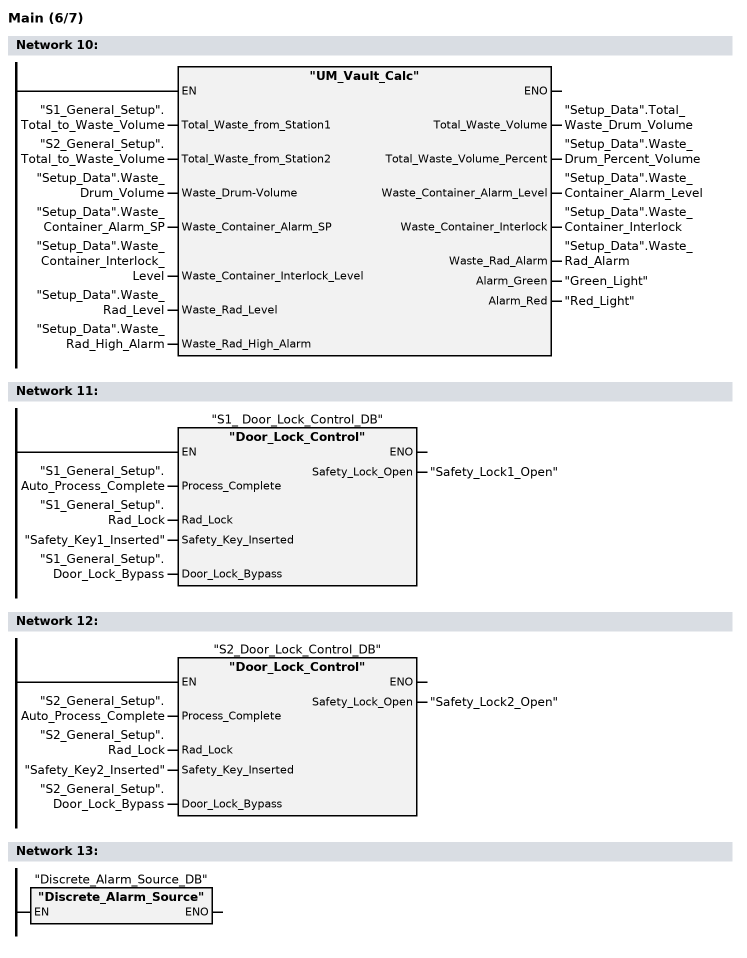
   RUNG wire#powerrail
      "UM_Vault_Calc"(Total_Waste_from_Station1 := "S1_General_Setup".Total_to_Waste_Volume, Total_Waste_from_Station2 := "S2_General_Setup".Total_to_Waste_Volume, "Waste_Drum-Volume" := "Setup_Data".Waste_Drum_Volume, Waste_Container_Alarm_SP := "Setup_Data".Waste_Container_Alarm_SP, Waste_Container_Interlock_Level := "Setup_Data".Waste_Container_Interlock_Level, Waste_Rad_Level := "Setup_Data".Waste_Rad_Level, Waste_Rad_High_Alarm := "Setup_Data".Waste_Rad_High_Alarm, Total_Waste_Volume => "Setup_Data".Total_Waste_Drum_Volume, Total_Waste_Volume_Percent => "Setup_Data".Waste_Drum_Percent_Volume, Waste_Container_Alarm_Level => "Setup_Data".Waste_Container_Alarm_Level, Waste_Container_Interlock => "Setup_Data".Waste_Container_Interlock, Waste_Rad_Alarm => "Setup_Data".Waste_Rad_Alarm, Alarm_Green => "Green_Light", Alarm_Red => "Red_Light")
   END_RUNG
   // the same network as SCL:
   "UM_Vault_Calc"(Total_Waste_from_Station1 := "S1_General_Setup".Total_to_Waste_Volume,
                   Total_Waste_from_Station2 := "S2_General_Setup".Total_to_Waste_Volume,
                   "Waste_Drum-Volume" := "Setup_Data".Waste_Drum_Volume,
                   Waste_Container_Alarm_SP := "Setup_Data".Waste_Container_Alarm_SP,
                   Waste_Container_Interlock_Level := "Setup_Data".Waste_Container_Interlock_Level,
                   Waste_Rad_Level := "Setup_Data".Waste_Rad_Level,
                   Waste_Rad_High_Alarm := "Setup_Data".Waste_Rad_High_Alarm,
                   Total_Waste_Volume => "Setup_Data".Total_Waste_Drum_Volume,
                   Total_Waste_Volume_Percent => "Setup_Data".Waste_Drum_Percent_Volume,
                   Waste_Container_Alarm_Level => "Setup_Data".Waste_Container_Alarm_Level,
                   Waste_Container_Interlock => "Setup_Data".Waste_Container_Interlock,
                   Waste_Rad_Alarm => "Setup_Data".Waste_Rad_Alarm,
                   Alarm_Green => "Green_Light",
                   Alarm_Red => "Red_Light");
END_REGION

REGION Network 11
   RUNG wire#powerrail
      "S1_ Door_Lock_Control_DB"(Process_Complete := "S1_General_Setup".Auto_Process_Complete, Rad_Lock := "S1_General_Setup".Rad_Lock, Safety_Key_Inserted := "Safety_Key1_Inserted", Door_Lock_Bypass := "S1_General_Setup".Door_Lock_Bypass, Safety_Lock_Open => "Safety_Lock1_Open")
   END_RUNG
   // the same network as SCL:
   "S1_ Door_Lock_Control_DB"(Process_Complete := "S1_General_Setup".Auto_Process_Complete,   // "Door_Lock_Control"
                           Rad_Lock := "S1_General_Setup".Rad_Lock,
                           Safety_Key_Inserted := "Safety_Key1_Inserted",
                           Door_Lock_Bypass := "S1_General_Setup".Door_Lock_Bypass,
                           Safety_Lock_Open => "Safety_Lock1_Open");
END_REGION

REGION Network 12
   RUNG wire#powerrail
      "S2_Door_Lock_Control_DB"(Process_Complete := "S2_General_Setup".Auto_Process_Complete, Rad_Lock := "S2_General_Setup".Rad_Lock, Safety_Key_Inserted := "Safety_Key2_Inserted", Door_Lock_Bypass := "S2_General_Setup".Door_Lock_Bypass, Safety_Lock_Open => "Safety_Lock2_Open")
   END_RUNG
   // the same network as SCL:
   "S2_Door_Lock_Control_DB"(Process_Complete := "S2_General_Setup".Auto_Process_Complete,   // "Door_Lock_Control"
                           Rad_Lock := "S2_General_Setup".Rad_Lock,
                           Safety_Key_Inserted := "Safety_Key2_Inserted",
                           Door_Lock_Bypass := "S2_General_Setup".Door_Lock_Bypass,
                           Safety_Lock_Open => "Safety_Lock2_Open");
END_REGION

REGION Network 13
   RUNG wire#powerrail
      "Discrete_Alarm_Source_DB"()
   END_RUNG
   // the same network as SCL:
   "Discrete_Alarm_Source_DB"();   // "Discrete_Alarm_Source"
END_REGION

REGION Network 14
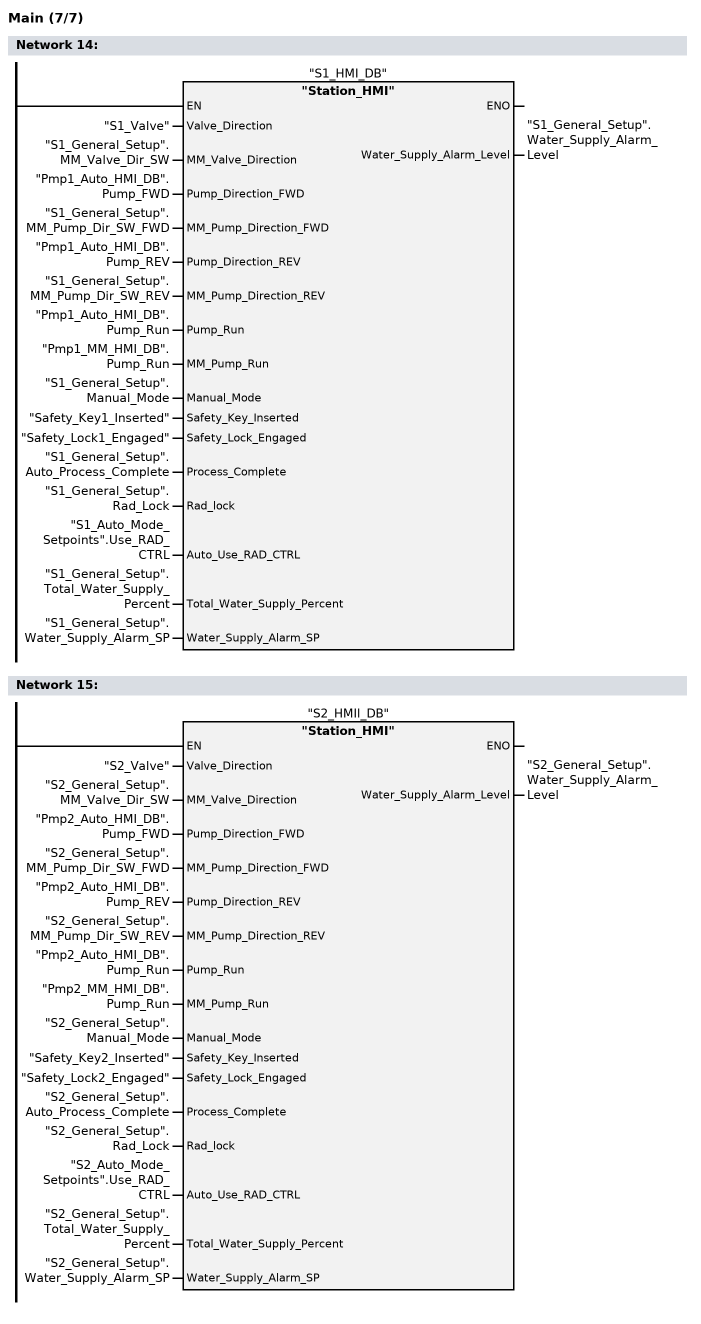
   RUNG wire#powerrail
      "S1_HMI_DB"(Valve_Direction := "S1_Valve", MM_Valve_Direction := "S1_General_Setup".MM_Valve_Dir_SW, Pump_Direction_FWD := "Pmp1_Auto_HMI_DB".Pump_FWD, MM_Pump_Direction_FWD := "S1_General_Setup".MM_Pump_Dir_SW_FWD, Pump_Direction_REV := "Pmp1_Auto_HMI_DB".Pump_REV, MM_Pump_Direction_REV := "S1_General_Setup".MM_Pump_Dir_SW_REV, Pump_Run := "Pmp1_Auto_HMI_DB".Pump_Run, MM_Pump_Run := "Pmp1_MM_HMI_DB".Pump_Run, Manual_Mode := "S1_General_Setup".Manual_Mode, Safety_Key_Inserted := "Safety_Key1_Inserted", Safety_Lock_Engaged := "Safety_Lock1_Engaged", Process_Complete := "S1_General_Setup".Auto_Process_Complete, Rad_lock := "S1_General_Setup".Rad_Lock, Auto_Use_RAD_CTRL := "S1_Auto_Mode_Setpoints".Use_RAD_CTRL, Total_Water_Supply_Percent := "S1_General_Setup".Total_Water_Supply_Percent, Water_Supply_Alarm_SP := "S1_General_Setup".Water_Supply_Alarm_SP, Water_Supply_Alarm_Level => "S1_General_Setup".Water_Supply_Alarm_Level)
   END_RUNG
   // the same network as SCL:
   "S1_HMI_DB"(Valve_Direction := "S1_Valve",   // "Station_HMI"
               MM_Valve_Direction := "S1_General_Setup".MM_Valve_Dir_SW,
               Pump_Direction_FWD := "Pmp1_Auto_HMI_DB".Pump_FWD,
               MM_Pump_Direction_FWD := "S1_General_Setup".MM_Pump_Dir_SW_FWD,
               Pump_Direction_REV := "Pmp1_Auto_HMI_DB".Pump_REV,
               MM_Pump_Direction_REV := "S1_General_Setup".MM_Pump_Dir_SW_REV,
               Pump_Run := "Pmp1_Auto_HMI_DB".Pump_Run,
               MM_Pump_Run := "Pmp1_MM_HMI_DB".Pump_Run,
               Manual_Mode := "S1_General_Setup".Manual_Mode,
               Safety_Key_Inserted := "Safety_Key1_Inserted",
               Safety_Lock_Engaged := "Safety_Lock1_Engaged",
               Process_Complete := "S1_General_Setup".Auto_Process_Complete,
               Rad_lock := "S1_General_Setup".Rad_Lock,
               Auto_Use_RAD_CTRL := "S1_Auto_Mode_Setpoints".Use_RAD_CTRL,
               Total_Water_Supply_Percent := "S1_General_Setup".Total_Water_Supply_Percent,
               Water_Supply_Alarm_SP := "S1_General_Setup".Water_Supply_Alarm_SP,
               Water_Supply_Alarm_Level => "S1_General_Setup".Water_Supply_Alarm_Level);
END_REGION

REGION Network 15
   RUNG wire#powerrail
      "S2_HMIl_DB"(Valve_Direction := "S2_Valve", MM_Valve_Direction := "S2_General_Setup".MM_Valve_Dir_SW, Pump_Direction_FWD := "Pmp2_Auto_HMI_DB".Pump_FWD, MM_Pump_Direction_FWD := "S2_General_Setup".MM_Pump_Dir_SW_FWD, Pump_Direction_REV := "Pmp2_Auto_HMI_DB".Pump_REV, MM_Pump_Direction_REV := "S2_General_Setup".MM_Pump_Dir_SW_REV, Pump_Run := "Pmp2_Auto_HMI_DB".Pump_Run, MM_Pump_Run := "Pmp2_MM_HMI_DB".Pump_Run, Manual_Mode := "S2_General_Setup".Manual_Mode, Safety_Key_Inserted := "Safety_Key2_Inserted", Safety_Lock_Engaged := "Safety_Lock2_Engaged", Process_Complete := "S2_General_Setup".Auto_Process_Complete, Rad_lock := "S2_General_Setup".Rad_Lock, Auto_Use_RAD_CTRL := "S2_Auto_Mode_Setpoints".Use_RAD_CTRL, Total_Water_Supply_Percent := "S2_General_Setup".Total_Water_Supply_Percent, Water_Supply_Alarm_SP := "S2_General_Setup".Water_Supply_Alarm_SP, Water_Supply_Alarm_Level => "S2_General_Setup".Water_Supply_Alarm_Level)
   END_RUNG
   // the same network as SCL:
   "S2_HMIl_DB"(Valve_Direction := "S2_Valve",   // "Station_HMI"
                MM_Valve_Direction := "S2_General_Setup".MM_Valve_Dir_SW,
                Pump_Direction_FWD := "Pmp2_Auto_HMI_DB".Pump_FWD,
                MM_Pump_Direction_FWD := "S2_General_Setup".MM_Pump_Dir_SW_FWD,
                Pump_Direction_REV := "Pmp2_Auto_HMI_DB".Pump_REV,
                MM_Pump_Direction_REV := "S2_General_Setup".MM_Pump_Dir_SW_REV,
                Pump_Run := "Pmp2_Auto_HMI_DB".Pump_Run,
                MM_Pump_Run := "Pmp2_MM_HMI_DB".Pump_Run,
                Manual_Mode := "S2_General_Setup".Manual_Mode,
                Safety_Key_Inserted := "Safety_Key2_Inserted",
                Safety_Lock_Engaged := "Safety_Lock2_Engaged",
                Process_Complete := "S2_General_Setup".Auto_Process_Complete,
                Rad_lock := "S2_General_Setup".Rad_Lock,
                Auto_Use_RAD_CTRL := "S2_Auto_Mode_Setpoints".Use_RAD_CTRL,
                Total_Water_Supply_Percent := "S2_General_Setup".Total_Water_Supply_Percent,
                Water_Supply_Alarm_SP := "S2_General_Setup".Water_Supply_Alarm_SP,
                Water_Supply_Alarm_Level => "S2_General_Setup".Water_Supply_Alarm_Level);
END_REGION
END_ORGANIZATION_BLOCK

(* ===== HMI "HMI_RT_1" =====
system functions are stored by id; their names below are inferred from use
connection "HMI_Connection_1": ETHERNET, S7_1500_OMS

HMI tags "Common tags"
   "Safety Relay Trip" : Bool = PLC Safety_Relay_Trip AT %I0.0, 1 s
   "CurrentUserName" : WString[10] AT %DB1.DBX0.0
   "CurrentGroupNum" : Int, internal
   "Total Waste Drum Volume" : Real = PLC Setup_Data.Total_Waste_Drum_Volume AT %DB1.DBD0, 1 s
   "Waste Drum Volume" : Real = PLC Setup_Data.Waste_Drum_Volume AT %DB1.DBD0, 1 s
   "Waste Drum Percent Volume" : Real = PLC Setup_Data.Waste_Drum_Percent_Volume AT %DB1.DBD0, 1 s
   "Waste Container Reset" : Bool = PLC Setup_Data.Waste_Container_Reset AT %DB1.DBD0, 1 s
   "Waste Drum Alarm Level" : Int = PLC Setup_Data.Waste_Container_Alarm_Level AT %DB1.DBD0, 1 s
   "Waste Drum Alarm SP" : Real = PLC Setup_Data.Waste_Container_Alarm_SP AT %DB1.DBD0, 1 s
   "Waste Rad High Alarm" : Real = PLC Setup_Data.Waste_Rad_High_Alarm AT %DB1.DBW0, 1 s
   "Waste Rad Level" : Real = PLC Setup_Data.Waste_Rad_Level AT %DB1.DBW0, 1 s
   "Waste Rad Alarm" : Bool = PLC Setup_Data.Waste_Rad_Alarm AT %DB1.DBD0, 1 s
   "Alarm Integer 1" : Int = PLC Discrete_Alarm_Source_DB.Alarm_Integer_1 AT %DB1.DBD0, 1 s
   "Pump 1 Data_Data_CMD_Trigger_Slew" : Bool = PLC Pmp1_Data.Data.CMD_Trigger.Slew AT %DB1.DBD0, 1 s
   "Waste Drum Level Interlock" : Real = PLC Setup_Data.Waste_Container_Interlock_Level, 1 s
   "Waste Drum Interlock" : Bool = PLC Setup_Data.Waste_Container_Interlock AT %DB1.DBD0, 1 s
   "Alarm Integer 2" : Int = PLC Discrete_Alarm_Source_DB.Alarm_Integer_2 AT %DB1.DBD0, 1 s
   "Estop Active" : Bool = PLC Setup_Data.Estop_Active AT %DB1.DBX0.0, 1 s
   "Buzzer Reset" : Bool = PLC Setup_Data.Buzzer_Reset AT %DB1.DBX0.0, 1 s
   "System Version" : String[254] = PLC Setup_Data.System_Version AT %DB1.DBD0, 1 s
   "UM Hi Level SW" : Bool = PLC UM_HI_Level_SW AT %I0.6, 1 s
   "Total Waste Drum Update" : Real = PLC S1_Automated_Run_DB.Auto_Mode_Instance.Total_Waste_Drum_Update AT %DB1.DBD0, 1 s
   "Waste Drum Update" : Bool = PLC S1_Automated_Run_DB.Auto_Mode_Instance.Waste_Drum_Update AT %DB1.DBX0.0, 1 s

HMI tags "Station 1"
   "Station 1 Door Close" : Int = PLC S1_HMI_DB.Door_Closed AT %DB1.DBW0, 1 s
   "Station 1 Door Locked" : Bool = PLC S1_HMI_DB.Door_Locked AT %I1.0, 1 s
   "Station 1 Auto Current Rinse Num" : Int = PLC S1_Automated_Run_DB.Auto_Current_Rinse_Number AT %DB1.DBW0, 1 s
   "Station 1 Auto Number of Rinses" : Int = PLC S1_Auto_Mode_Setpoints.Number_of_Rinses AT %DB1.DBX0.0, 1 s
   "Station 1 Auto Process State" : String[254] = PLC S1_Automated_Run_DB.Auto_Current_Process_State AT %DB1.DBW0, 1 s
   "Station 1 Run State" : Int = PLC S1_Automated_Run_DB.Run_State AT %DB1.DBW0, 1 s
   "Station 1 Hide Vessel Tubing" : Bool = PLC S1_HMI_DB.Hide_Vessel_Tubing AT %DB1.DBX0.0, 1 s
   "Station 1 PMP FWD" : Bool = PLC S1_HMI_DB.Display_PMP_FWD AT %DB1.DBX0.0, 1 s
   "Station 1 PMP REV" : Bool = PLC S1_HMI_DB.Display_PMP_REV AT %DB1.DBX0.0, 1 s
   "Station 1 Pump Run" : Bool = PLC Pmp1_Auto_HMI_DB.Pump_Run, 1 s
   "Station 1 Pump Tubing" : Int = PLC S1_HMI_DB.Tubing_Pump, 1 s
   "Station 1 Recycle Mode" : String[254] = PLC S1_HMI_DB.Recycle_Mode_HMI, 1 s
   "Station 1 Rad Interlock" : Bool = PLC S1_General_Setup.Rad_Lock, 1 s
   "Station 1 Tubing Rinse" : Int = PLC S1_HMI_DB.Tubing_Rinse AT %DB1.DBW0, 1 s
   "Station 1 Tubing Drain" : Int = PLC S1_HMI_DB.Tubing_Drain AT %DB1.DBW0, 1 s
   "Station 1 Valve Pump" : Int = PLC S1_HMI_DB.Valve_Pump AT %DB1.DBW0, 1 s
   "Station 1 Valve Rinse" : Int = PLC S1_HMI_DB.Valve_Rinse AT %DB1.DBX0.0, 1 s
   "Station 1 Valve Drain" : Int = PLC S1_HMI_DB.Valve_Drain AT %DB1.DBX0.0, 1 s
   "Station 1 Tubing Vessel" : Int = PLC S1_HMI_DB.Tubing_Vessel AT %DB1.DBW0, 1 s
   "Station 1 Estop PB Active" : Bool = PLC Estop1_PB_Active AT %I1.4, 1 s
   "Station 1 Pump Speed SP RPM" : Real = PLC S1_General_Setup.Man_Speed_SP, 1 s
   "Station 1 MM Pump Dir FWD" : Bool = PLC S1_General_Setup.MM_Pump_Dir_SW_FWD AT %DB1.DBX0.0, 1 s
   "Station 1 MM Valve Direction SW" : Bool = PLC S1_General_Setup.MM_Valve_Dir_SW, 1 s
   "Station 1 Process Running" : Bool = PLC S1_Automated_Run_DB.Process_Running, 1 s
   "Station 1 Door Lock Open" : Bool = PLC S1_General_Setup.Door_Lock_Bypass AT %DB1.DBX0.0, 1 s
   "Station 1 Auto Process Complete" : Bool = PLC S1_General_Setup.Auto_Process_Complete, 1 s
   "Station 1 Door Lock Bypass" : Bool = PLC S1_HMI_DB.Door_Lock_Bypass_HMI, 1 s
   "Station 1 Rad Lock Bypass" : Bool = PLC S1_General_Setup.Rad_Lock_Bypass AT %DB1.DBX0.0, 1 s
   "Station 1 RAD Complete Rinses" : Int = PLC S1_Automated_Run_DB.Auto_Mode_Instance.RAD_Complete_Rinses AT %DB1.DBW0, 1 s
   "Station 1 Auto Info" : Int = PLC S1_HMI_DB.Auto_Info_HMI AT %DB1.DBW0, 1 s
   "Station 1 Vessel Rad Alarm" : Bool = PLC S1_Interlocks_DB.Vessel_Rad_Alarm AT %DB1.DBX0.0, 1 s
   "Station 1 Pump Rad Alarm" : Bool = PLC S1_Interlocks_DB.Pump_Rad_Alarm AT %DB1.DBX0.0, 1 s
   "Station 1 Manual Mode" : Bool = PLC S1_General_Setup.Manual_Mode, 1 s
   "S1 Setup Data_Leave Manual Screen" : Bool = PLC S1_General_Setup.Leave_Manual_Screen, 1 s
   "Station 1 Container Water Supply Volume" : Real = PLC S1_General_Setup.Container_Water_Supply_Volume AT %DB1.DBD0, 1 s
   "Station 1 Total Water Supply Volume" : Real = PLC S1_General_Setup.Total_Water_Supply_Volume AT %DB1.DBD0, 1 s
   "Station 1 Total Water Supply Percent" : Real = PLC S1_General_Setup.Total_Water_Supply_Percent AT %DB1.DBX0.0, 1 s
   "Station 1 New Water Container" : Bool = PLC S1_General_Setup.New_Water_Container AT %DB1.DBX0.0, 1 s
   "Station 1 New Waste Container" : Bool = PLC S1_General_Setup.New_Waste_Container AT %DB1.DBX0.0, 1 s
   "Station 1 Water Supply Alarm SP" : Real = PLC S1_General_Setup.Water_Supply_Alarm_SP AT %DB1.DBX0.0, 1 s
   "Station 1 Water Supply Alarm Level" : Int = PLC S1_General_Setup.Water_Supply_Alarm_Level AT %DB1.DBX0.0, 1 s
   "Station 1 Warning 1" : Bool = PLC S1_HMI_DB.Warning_1 AT %DB1.DBD0, 1 s
   "Station 1 Warning 2" : Bool = PLC S1_HMI_DB.Warning_2 AT %DB1.DBX0.0, 1 s
   "Station 1 MM Pump Dir REV" : Bool = PLC S1_General_Setup.MM_Pump_Dir_SW_REV AT %DB1.DBX0.0, 1 s
   "Station 1 MM Pump Slew PB" : Bool = PLC S1_General_Setup.MM_Pump_Slew_PB AT %DB1.DBX0.0, 1 s
   "Pump 1 Motor_Reset" : Bool = PLC Pmp1_Data.Data.Reset AT %DB1.DBD0, 1 s
   "Station 1 MM PMP FWD" : Bool = PLC Pmp1_MM_HMI_DB.Pump_FWD AT %DB1.DBX0.0, 1 s
   "Station 1 MM PMP REV" : Bool = PLC Pmp1_MM_HMI_DB.Pump_REV AT %DB1.DBX0.0, 1 s
   "Station 1 MM PMP Run" : Bool = PLC Pmp1_MM_HMI_DB.Pump_Run AT %DB1.DBX0.0, 1 s
   "Station 1 Water Supply Interlock SP" : Real = PLC S1_General_Setup.Water_Supply_Interlock_Level, 1 s
   "Station 1 Water Supply Interlock" : Bool = PLC S1_General_Setup.Water_Supply_Interlock AT %DB1.DBD0, 1 s
   "Station 1 Pump Error Code" : UInt = PLC S1_General_Setup.Pump_Error_Code AT %DB1.DBW0, 1 s
   "Station 1 Pump Error Code Bit" : Bool = PLC S1_General_Setup.Pump_Error_Bit AT %DB1.DBX0.0, 1 s
   "Station 1 MM Feedback RPM" : Real = PLC S1_General_Setup.MM_Feedback_RPM AT %DB1.DBD0, 1 s
   "Station 1 Total Water Supply Update" : Real = PLC S1_Automated_Run_DB.Auto_Mode_Instance.Total_Water_Supply_Update AT %DB1.DBD0, 1 s
   "Station 1 Water Update" : Bool = PLC S1_Automated_Run_DB.Auto_Mode_Instance.Water_Update AT %DB1.DBX0.0, 1 s

HMI tags "Station 1 Setup"
   "S1 Auto Pump Drain Max Speed" : Real = PLC S1_Auto_Mode_Setpoints.Pump_Drain_Full_Speed, 1 s
   "S1 Auto Ramp Drain Step" : Int = PLC S1_Auto_Mode_Setpoints.Ramp_Drain_Step AT %DB1.DBW0, 1 s
   "S1 Auto Ramp Drain Time" : Time = PLC S1_Auto_Mode_Setpoints.Ramp_Drain_Time AT %DB1.DBD0, 1 s
   "S1 Auto Pump Rinse Max Speed" : Real = PLC S1_Auto_Mode_Setpoints.Pump_Rinse_Full_Speed AT %DB1.DBW0, 1 s
   "S1 Auto Ramp Rinse Step" : Int = PLC S1_Auto_Mode_Setpoints.Ramp_Rinse_Step AT %DB1.DBW0, 1 s
   "S1 Auto Ramp Rinse Time" : Time = PLC S1_Auto_Mode_Setpoints.Ramp_Rinse_Time AT %DB1.DBD0, 1 s
   "S1 Auto Drain Run Time" : Time = PLC S1_Auto_Mode_Setpoints.Run_Drain_Time AT %DB1.DBD0, 1 s
   "S1 Auto Rinse Run Time" : Time = PLC S1_Auto_Mode_Setpoints.Run_Rinse_Time AT %DB1.DBD0, 1 s
   "S1 Auto Number of Rinses" : Int = PLC S1_Auto_Mode_Setpoints.Number_of_Rinses AT %DB1.DBW0, 1 s
   "S1 Auto Use RAD CTRL" : Bool = PLC S1_Auto_Mode_Setpoints.Use_RAD_CTRL AT %DB1.DBX0.0, 1 s
   "S1 Auto Rinse to RAD Level" : Real = PLC S1_Auto_Mode_Setpoints.Rinse_to_RAD_Level AT %DB1.DBW0, 1 s
   "S1 Pump Factor" : Real = PLC S1_General_Setup.Pump_Factor AT %DB1.DBX0.0, 1 s
   "S1 Pump Stroke Volume" : Real = PLC S1_General_Setup.Pump_Stroke_Volume AT %DB1.DBD0, 1 s
   "S1 Auto Pump Remove Max Speed" : Real = PLC S1_Auto_Mode_Setpoints.Pump_Remove_Full_Speed AT %DB1.DBD0, 1 s
   "S1Auto Ramp Remove Step" : Int = PLC S1_Auto_Mode_Setpoints.Ramp_Remove_Step AT %DB1.DBW0, 1 s
   "S1Auto Ramp Remove Time" : Time = PLC S1_Auto_Mode_Setpoints.Ramp_Remove_Time AT %DB1.DBD0, 1 s
   "S1 Auto Remove Run Time" : Time = PLC S1_Auto_Mode_Setpoints.Run_Remove_Time AT %DB1.DBD0, 1 s

HMI tags "Station 1 RAD Levels"
   "Station 1 Pump Rad Alarm Level" : Real = PLC S1_General_Setup.Pump_Alarm_Level AT %DB1.DBW0, 1 s
   "Station 1 Pump Rad Level" : Real = PLC S1_General_Setup.Pump_Rad_Level AT %DB1.DBD0, 1 s
   "Station 1 Vessel Rad Alarm Level" : Real = PLC S1_General_Setup.Vessel_Alarm_Level AT %DB1.DBW0, 1 s
   "Station 1 Vessel Rad Level" : Real = PLC S1_General_Setup.Vessel_Rad_Level AT %DB1.DBW0, 1 s

HMI tags "Station 2 RAD Levels"
   "Station 2 Pump Rad Alarm Level" : Real = PLC S2_General_Setup.Pump_Alarm_Level AT %DB1.DBW0, 1 s
   "Station 2 Pump Rad Level" : Real = PLC S2_General_Setup.Pump_Rad_Level AT %DB1.DBD0, 1 s
   "Station 2 Vessel Rad Alarm Level" : Real = PLC S2_General_Setup.Vessel_Alarm_Level AT %DB1.DBW0, 1 s
   "Station 2 Vessel Rad Level" : Real = PLC S2_General_Setup.Vessel_Rad_Level AT %DB1.DBW0, 1 s

HMI tags "Station 2 Setup"
   "S2 Auto Pump Drain Max Speed" : Real = PLC S2_Auto_Mode_Setpoints."Pump_Drain_Full Speed", 1 s
   "S2 Auto Ramp Drain Step" : Int = PLC S2_Auto_Mode_Setpoints.Ramp_Drain_Step AT %DB1.DBW0, 1 s
   "S2 Auto Ramp Drain Time" : Time = PLC S2_Auto_Mode_Setpoints.Ramp_Drain_Time AT %DB1.DBD0, 1 s
   "S2 Auto Pump Rinse Max Speed" : Real = PLC S2_Auto_Mode_Setpoints.Pump_Rinse_Full_Speed AT %DB1.DBW0, 1 s
   "S2 Auto Ramp Rinse Step" : Int = PLC S2_Auto_Mode_Setpoints.Ramp_Rinse_Step AT %DB1.DBW0, 1 s
   "S2 Auto Ramp Rinse Time" : Time = PLC S2_Auto_Mode_Setpoints.Ramp_Rinse_Time AT %DB1.DBD0, 1 s
   "S2 Auto Drain Run Time" : Time = PLC S2_Auto_Mode_Setpoints.Run_Drain_Time AT %DB1.DBD0, 1 s
   "S2 Auto Rinse Run Time" : Time = PLC S2_Auto_Mode_Setpoints.Run_Rinse_Time AT %DB1.DBD0, 1 s
   "S2 Auto Number of Rinses" : Int = PLC S2_Auto_Mode_Setpoints.Number_of_Rinses AT %DB1.DBW0, 1 s
   "S2 Auto Use RAD CTRL" : Bool = PLC S2_Auto_Mode_Setpoints.Use_RAD_CTRL AT %DB1.DBX0.0, 1 s
   "S2 Auto Rinse to RAD Level" : Real = PLC S2_Auto_Mode_Setpoints.Rinse_to_RAD_Level AT %DB1.DBW0, 1 s
   "S2 Pump Factor" : Real = PLC S2_General_Setup.Pump_Factor AT %DB1.DBX0.0, 1 s
   "S2 Pump Stroke Volume" : Real = PLC S2_General_Setup.Pump_Stroke_Volume AT %DB1.DBD0, 1 s
   "S2 Auto Ramp Remove Step" : Int = PLC S2_Auto_Mode_Setpoints.Ramp_Remove_Step AT %DB1.DBW0, 1 s
   "S2 Auto Ramp Remove Time" : Time = PLC S2_Auto_Mode_Setpoints.Ramp_Remove_Time AT %DB1.DBD0, 1 s
   "S2 Auto Pump Remove Max Speed" : Real = PLC S2_Auto_Mode_Setpoints.Pump_Remove_Full_Speed AT %DB1.DBD0, 1 s
   "S2 Auto Remove Run Time" : Time = PLC S2_Auto_Mode_Setpoints.Run_Remove_Time AT %DB1.DBD0, 1 s

HMI tags "Station 2"
   "Station 2 Manual Mode" : Bool = PLC S2_General_Setup.Manual_Mode, 1 s
   "Station 2 Process Running" : Bool = PLC S2_Automated_Run_DB.Process_Running, 1 s
   "Station 2 MM Pump Dir FWD" : Bool = PLC S2_General_Setup.MM_Pump_Dir_SW_FWD AT %DB1.DBX0.0, 1 s
   "Station 2 MM Valve Direction SW" : Bool = PLC S2_General_Setup.MM_Valve_Dir_SW, 1 s
   "Station 2 Run State" : Int = PLC S2_Automated_Run_DB.Run_State AT %DB1.DBW0, 1 s
   "Station 2 Pump Tubing" : Int = PLC S2_HMIl_DB.Tubing_Pump, 1 s
   "Station 2 Tubing Rinse" : Int = PLC S2_HMIl_DB.Tubing_Rinse AT %DB1.DBW0, 1 s
   "Station 2 Tubing Drain" : Int = PLC S2_HMIl_DB.Tubing_Drain AT %DB1.DBW0, 1 s
   "Station 2 Valve Rinse" : Int = PLC S2_HMIl_DB.Valve_Rinse AT %DB1.DBX0.0, 1 s
   "Station 2 Valve Drain" : Int = PLC S2_HMIl_DB.Valve_Drain AT %DB1.DBX0.0, 1 s
   "Station 2 Valve Pump" : Int = PLC S2_HMIl_DB.Valve_Pump AT %DB1.DBW0, 1 s
   "Station 2 PMP FWD" : Bool = PLC S2_HMIl_DB.Display_PMP_FWD AT %DB1.DBX0.0, 1 s
   "Station 2 PMP REV" : Bool = PLC S2_HMIl_DB.Display_PMP_REV AT %DB1.DBX0.0, 1 s
   "Station 2 Door Lock Open" : Bool = PLC S2_General_Setup.Door_Lock_Bypass AT %DB1.DBX0.0, 1 s
   "Station 2 Rad Lock Bypass" : Bool = PLC S2_General_Setup.Rad_Lock_Bypass AT %DB1.DBX0.0, 1 s
   "S2 Setup Data_Leave Manual Screen" : Bool = PLC S2_General_Setup.Leave_Manual_Screen, 1 s
   "Station 2 Rad Interlock" : Bool = PLC S2_General_Setup.Rad_Lock AT %DB1.DBX0.0, 1 s
   "Station 2 Estop PB Active" : Bool = PLC Estop2_PB_Active AT %I1.5, 1 s
   "Station 2 Auto Process Complete" : Bool = PLC S2_General_Setup.Auto_Process_Complete AT %DB1.DBX0.0, 1 s
   "Station 2 Door Close" : Int = PLC S2_HMIl_DB.Door_Closed AT %DB1.DBX0.0, 1 s
   "Station 2 Door Locked" : Bool = PLC S2_HMIl_DB.Door_Locked AT %DB1.DBX0.0, 1 s
   "Station 2 Auto Current Rinse Num" : Int = PLC S2_Automated_Run_DB.Auto_Current_Rinse_Number AT %DB1.DBW0, 1 s
   "Station 2 Auto Number of Rinses" : Int = PLC S2_Auto_Mode_Setpoints.Number_of_Rinses AT %DB1.DBW0, 1 s
   "Station 2 Auto Process State" : String[254] = PLC S2_Automated_Run_DB.Auto_Current_Process_State AT %DB1.DBW0, 1 s
   "Station 2 Hide Vessel Tubing" : Bool = PLC S2_HMIl_DB.Hide_Vessel_Tubing AT %DB1.DBX0.0, 1 s
   "Station 2 Recycle Mode" : String[254] = PLC S2_HMIl_DB.Recycle_Mode_HMI AT %DB1.DBX0.0, 1 s
   "Station 2 Tubing Vessel" : Int = PLC S2_HMIl_DB.Tubing_Vessel AT %DB1.DBX0.0, 1 s
   "Station 2 Door Lock Bypass" : Bool = PLC S2_HMIl_DB.Door_Lock_Bypass_HMI AT %DB1.DBX0.0, 1 s
   "Station 2 RAD Complete Rinses" : Int = PLC S2_Automated_Run_DB.Auto_Mode_Instance.RAD_Complete_Rinses AT %DB1.DBX0.0, 1 s
   "Station 2 Auto Info" : Int = PLC S2_HMIl_DB.Auto_Info_HMI AT %DB1.DBW0, 1 s
   "Station 2 Vessel Rad Alarm" : Bool = PLC S2_Interlocks_DB.Vessel_Rad_Alarm AT %DB1.DBW0, 1 s
   "Station 2 Pump Rad Alarm" : Bool = PLC S2_Interlocks_DB.Pump_Rad_Alarm AT %DB1.DBW0, 1 s
   "Station 2 Container Water Supply Volume" : Real = PLC S2_General_Setup.Container_Water_Supply_Volume AT %DB1.DBD0, 1 s
   "Station 2 Total Water Supply Volume" : Real = PLC S2_General_Setup.Total_Water_Supply_Volume AT %DB1.DBD0, 1 s
   "Station 2 Total Water Supply Percent" : Real = PLC S2_General_Setup.Total_Water_Supply_Percent AT %DB1.DBD0, 1 s
   "Station 2 New Water Container" : Bool = PLC S2_General_Setup.New_Water_Container AT %DB1.DBX0.0, 1 s
   "Station 2 New Waste Container" : Bool = PLC S2_General_Setup.New_Waste_Container AT %DB1.DBX0.0, 1 s
   "Station 2 Water Supply Alarm SP" : Real = PLC S2_General_Setup.Water_Supply_Alarm_SP AT %DB1.DBX0.0, 1 s
   "Station 2 Water Supply Alarm Level" : Int = PLC S2_General_Setup.Water_Supply_Alarm_Level AT %DB1.DBX0.0, 1 s
   "Station 2 MM Pump Dir REV" : Bool = PLC S2_General_Setup.MM_Pump_Dir_SW_REV AT %DB1.DBD0, 1 s
   "Station 2 MM Pump Slew PB" : Bool = PLC S2_General_Setup.MM_Pump_Slew_PB AT %DB1.DBX0.0, 1 s
   "Station 2 MM Pump Run" : Bool = PLC Pmp2_MM_HMI_DB.Pump_Run AT %DB1.DBX0.0, 1 s
   "Station 2 MM Pump FWD" : Bool = PLC Pmp2_MM_HMI_DB.Pump_FWD AT %DB1.DBX0.0, 1 s
   "Station 2 MM Pump REV" : Bool = PLC Pmp2_MM_HMI_DB.Pump_REV AT %DB1.DBX0.0, 1 s
   "Station 2 Pump Speed RPM SP" : Real = PLC S2_General_Setup.Man_Speed_SP AT %DB1.DBX0.0, 1 s
   "Pump 2 Motor_Reset" : Bool = PLC Pmp2_Data.Data.Reset AT %DB1.DBD0, 1 s
   "Station 2 Warning 1" : Bool = PLC S2_HMIl_DB.Warning_1 AT %DB1.DBX0.0, 1 s
   "Station 2 Warning 2" : Bool = PLC S2_HMIl_DB.Warning_2 AT %DB1.DBX0.0, 1 s
   "Station 2 Pump Run" : Bool = PLC Pmp2_Auto_HMI_DB.Pump_Run AT %DB1.DBX0.0, 1 s
   "Station 2 Water Supply Interlock SP" : Real = PLC S2_General_Setup.Water_Supply_Interlock_Level, 1 s
   "Station 2 Water Supply Interlock" : Bool = PLC S2_General_Setup.Water_Supply_Interlock AT %DB1.DBD0, 1 s
   "Station 2 Pump Error Code" : UInt = PLC S2_General_Setup.Pump_Error_Code AT %DB1.DBD0, 1 s
   "Station 2 Pump Error Code Bit" : Bool = PLC S2_General_Setup.Pump_Error_Bit AT %DB1.DBD0, 1 s
   "Station 2 MM Feedback RPM" : Real = PLC S2_General_Setup.MM_Feedback_RPM AT %DB1.DBD0, 1 s
   "Station 2 Total Water Supply Update" : Real = PLC S2_Automated_Run_DB.Auto_Mode_Instance.Total_Water_Supply_Update AT %DB1.DBD0, 1 s
   "Station 2 Water Update" : Bool = PLC S2_Automated_Run_DB.Auto_Mode_Instance.Water_Update AT %DB1.DBX0.0, 1 s

discrete alarms
   1: 'Station 1 Estop Active', class Errors, trigger "Alarm Integer 1" bit 0
   2: 'Station 2 Estop Active', class Errors, trigger "Alarm Integer 1" bit 1
   3: 'Safety Relay Tripped', class Errors, trigger "Alarm Integer 1" bit 2
   4: 'Station 1 Radiation Lock Active', class Errors, trigger "Alarm Integer 1" bit 3
   5: 'Station 2 Radiation Lock Active', class Errors, trigger "Alarm Integer 1" bit 4
   6: 'Station 1 Rad Lock Bypass', class Warnings, trigger "Alarm Integer 1" bit 5
   7: 'Station 2 Rad Lock Bypass', class Warnings, trigger "Alarm Integer 1" bit 6
   8: 'Station 1 Door Lock Bypass', class Warnings, trigger "Alarm Integer 1" bit 7
   9: 'Station 2 Door Lock Bypass', class Warnings, trigger "Alarm Integer 1" bit 8
   10: 'New Unwanted Material Container', class Warnings, trigger "Alarm Integer 1" bit 9
   11: 'Station 1 New Water Container', class Warnings, trigger "Alarm Integer 1" bit 10
   12: 'Station 2 New Water Container', class Warnings, trigger "Alarm Integer 1" bit 11
   13: 'Station 1 Water Container Low Interlock', class Errors, trigger "Alarm Integer 1" bit 12
   15: 'UM Container High Interlock', class Errors, trigger "Alarm Integer 1" bit 14
   14: 'Station 2 Water Container Low Interlock', class Errors, trigger "Alarm Integer 1" bit 13
   17: 'Pump 1 Motor Error', class Warnings, trigger "Alarm Integer 2" bit 0
   18: 'Pump 2 Motor Error', class Warnings, trigger "Alarm Integer 2" bit 1
   16: 'UM Safety High Level', class Errors, trigger "Alarm Integer 2" bit 2
   19: 'Station 1 Pump Failure', class Errors, trigger "Alarm Integer 2" bit 3
   20: 'Station 2 Pump Failure', class Errors, trigger "Alarm Integer 2" bit 4

analog alarms
   1: 'Station 1 Pump Cave RAD High', class Errors, trigger "Station 1 Pump Rad Level"
   2: 'UM Container Level High', class Errors, trigger "Waste Drum Alarm Level"
   3: 'Station 1 Vessel Cave RAD High', class Errors, trigger "Station 1 Vessel Rad Level"
   4: 'Station 2 Pump Cave RAD High', class Errors, trigger "Station 2 Pump Rad Level"
   5: 'Station 2 Vessel Cave RAD High', class Errors, trigger "Station 2 Vessel Rad Level"
   6: 'Waste Vault RAD High', class Errors, trigger "Waste Rad Level"
   7: 'Station 1 Water Supply Low', class Errors, trigger "Station 1 Water Supply Alarm Level"
   8: 'Station 2 Water Supply Low', class Errors, trigger "Station 2 Water Supply Alarm Level"

screen "Home Screen" 1280x700, template "Navigation"
   Rectangle "Rectangle_1" at 208,8 size 443x662
      Appearance <- "Station 1 Run State"
   Rectangle "Rectangle_31" at 796,8 size 440x662
      Appearance <- "Station 2 Run State"
   Group "Group_1" at 252,480 size 114x111
   Group "Group_2" at 220,135 size 170x31; Text 'SYSTEM 1'
   TextField "Text field_3" at 415,370 size 113x25; Text 'PUMP CAVE'
   SymbolLibrary "Symbol library_2" at 281,208 size 10x33
      Appearance <- "Station 1 Tubing Rinse"
   SymbolLibrary "Symbol library_5" at 547,491 size 15x16
      Appearance <- "Station 1 Tubing Vessel"
   SymbolLibrary "Symbol library_6" at 553,217 size 10x84
      Appearance <- "Station 1 Pump Tubing"
   TextField "Text field_8" at 220,81 size 64x27; Text 'MODE:'
   IOField "I/O field_1" at 281,81 size 149x28; FormatPattern ??????????
      ProcessValue <- "Station 1 Recycle Mode"
   TextField "Text field_9" at 220,127 size 120x39; Text 'ACTIVE'
      Visibility <- "Station 1 Run State"
   TextField "Text field_10" at 220,127 size 86x39; Text 'STOP'
      Visibility <- "Station 1 Run State"
   IOField "I/O field_2" at 372,105 size 108x29; FormatPattern ????????
      ProcessValue <- "Station 1 Auto Process State"
   TextField "Text field_11" at 221,106 size 152x27; Text 'PROCESS STATE:'
   Group "Group_3" at 222,35 size 177x42; Text 'SYSTEM 1'
   SymbolLibrary "Symbol library_9" at 553,479 size 10x18
      Appearance <- "Station 1 Tubing Vessel"
   TextField "Text field_13" at 670,426 size 114x25; Text 'UNWANTED'
   TextField "Text field_14" at 251,378 size 75x23; Text 'SUPPLY'
   TextField "Text field_15" at 253,363 size 71x23; Text 'WATER'
   Group "Group_6" at 436,483 size 49x85
   Group "Group_10" at 246,431 size 123x173
      HorizontalMovement <- "Station 1 Door Close"
   TextField "Text field_16" at 422,408 size 80x25; Text 'LOCKED'
      Visibility <- "Station 1 Door Locked"
   SymbolLibrary "Symbol library_18" at 456,498 size 97x10
      Visibility <- "Station 1 Hide Vessel Tubing"
      Appearance <- "Station 1 Tubing Vessel"
   Group "Group_12" at 485,32 size 153x83
   Switch "Pushbutton_Emergency_2" at 415,35 size 60x61; CaptionText 'Switch'; TextOff '0'; TextOn '1'; PictureOff "Pushbutton_Emergency_Off_256c"; PictureOn "Pushbutton_Emergency_On_256c"
      Visibility <- "Station 1 Estop PB Active"
      ProcessValue <- "Station 1 Estop PB Active"
   TextField "Text field_20" at 413,13 size 65x25; Text 'ESTOP'
      Visibility <- "Station 1 Estop PB Active"
   TextField "Text field_21" at 404,601 size 128x25; Text 'VESSEL CAVE'
   Group "Group_13" at 485,33 size 153x132
   GraphicView "Graphic view_2" at 437,517 size 46x48; Picture "Graphic_1"
      Visibility <- "Station 1 Vessel Rad Alarm"
   Bar "Bar_1" at 691,249 size 66x109; MinimumValue 0; MaximumValue 100
      ProcessValue <- "Total Waste Drum Volume"
      MaximumValue <- "Waste Drum Volume"
   SymbolLibrary "Symbol library_21" at 688,242 size 71x124
   GraphicView "Graphic view_3" at 700,101 size 42x43; Picture "Graphic_1"
      Visibility <- "Waste Rad Alarm"
   SymbolLibrary "Symbol library_24" at 566,201 size 149x10
      Appearance <- "Station 1 Tubing Drain"
   SymbolLibrary "Symbol library_30" at 258,226 size 59x105
   Bar "Bar_2" at 258,248 size 59x79; MinimumValue 0; MaximumValue 100
      Appearance <- "Station 1 Water Supply Alarm Level"
      ProcessValue <- "Station 1 Total Water Supply Volume"
      MaximumValue <- "Station 1 Container Water Supply Volume"
   IOField "I/O field_15" at 663,385 size 122x33; FormatPattern 999.9; Unit  %
      ProcessValue <- "Waste Drum Percent Volume"
      Appearance <- "Waste Drum Alarm Level"
   SymbolLibrary "Symbol library_3" at 712,215 size 9x30
      Appearance <- "Station 1 Tubing Drain"
   SymbolLibrary "Symbol library_4" at 706,202 size 14x15
      Appearance <- "Station 1 Tubing Drain"
   SymbolLibrary "Symbol library_1" at 282,202 size 14x14
      Appearance <- "Station 1 Tubing Rinse"
   IOField "I/O field_16" at 237,332 size 100x33; FormatPattern 999.9; Unit  %
      ProcessValue <- "Station 1 Total Water Supply Percent"
      Appearance <- "Station 1 Water Supply Alarm Level"
   SymbolLibrary "Symbol library_7" at 290,201 size 260x10
      Appearance <- "Station 1 Tubing Rinse"
   Group "Group" at 540,184 size 37x41
   Group "Group_4" at 401,217 size 123x33
   SymbolLibrary "Symbol library_8" at 553,278 size 10x209
      Appearance <- "Station 1 Pump Tubing"
   SymbolLibrary "Symbol library_16" at 399,253 size 159x73
   GraphicView "Graphic view_1" at 433,263 size 46x48; Picture "Graphic_1"
      Visibility <- "Station 1 Pump Rad Alarm"
   Group "Group_16" at 808,134 size 170x31; Text 'SYSTEM 1'
   TextField "Text field_36" at 919,370 size 113x25; Text 'PUMP CAVE'
   SymbolLibrary "Symbol library_29" at 1148,210 size 10x50
      Appearance <- "Station 2 Tubing Rinse"
   SymbolLibrary "Symbol library_32" at 1142,203 size 14x15
      Appearance <- "Station 2 Tubing Rinse"
   SymbolLibrary "Symbol library_33" at 871,490 size 14x16
      Appearance <- "Station 2 Tubing Vessel"
   TextField "Text field_41" at 808,80 size 64x27; Text 'MODE:'
   IOField "I/O field_18" at 868,80 size 141x28; FormatPattern ??????????
      ProcessValue <- "Station 2 Recycle Mode"
   TextField "Text field_42" at 808,126 size 120x39; Text 'ACTIVE'
      Visibility <- "Station 2 Run State"
   TextField "Text field_43" at 810,126 size 86x39; Text 'STOP'
      Visibility <- "Station 2 Run State"
   IOField "I/O field_19" at 964,104 size 108x29; FormatPattern ????????
      ProcessValue <- "Station 2 Auto Process State"
   TextField "Text field_44" at 809,105 size 152x27; Text 'PROCESS STATE:'
   Group "Group_18" at 810,34 size 177x42; Text 'SYSTEM 1'
   SymbolLibrary "Symbol library_47" at 724,202 size 15x15
      Appearance <- "Station 2 Tubing Drain"
   SymbolLibrary "Symbol library_48" at 731,201 size 129x10
      Appearance <- "Station 2 Tubing Drain"
   SymbolLibrary "Symbol library_53" at 723,212 size 10x32
      Appearance <- "Station 2 Tubing Drain"
   Group "Group_17" at 907,218 size 123x33
   SymbolLibrary "Symbol library_12" at 889,202 size 261x10
      Appearance <- "Station 2 Tubing Rinse"
   TextField "Text field_46" at 1120,378 size 75x23; Text 'SUPPLY'
   TextField "Text field_67" at 1123,362 size 71x23; Text 'WATER'
   SymbolLibrary "Symbol library_22" at 1124,225 size 59x105
   Bar "Bar_3" at 1124,247 size 59x79; MinimumValue 0; MaximumValue 100
      Appearance <- "Station 2 Water Supply Alarm Level"
      ProcessValue <- "Station 2 Total Water Supply Volume"
      MaximumValue <- "Station 2 Container Water Supply Volume"
   IOField "I/O field_17" at 1105,331 size 100x33; FormatPattern 999.9; Unit  %
      ProcessValue <- "Station 2 Total Water Supply Percent"
      Appearance <- "Station 2 Water Supply Alarm Level"
   Group "Group_21" at 947,482 size 49x85
   TextField "Text field_49" at 933,407 size 80x25; Text 'LOCKED'
      Visibility <- "Station 2 Door Locked"
   TextField "Text field_54" at 915,600 size 128x25; Text 'VESSEL CAVE'
   GraphicView "Graphic view_6" at 948,516 size 46x48; Picture "Graphic_1"
      Visibility <- "Station 2 Vessel Rad Alarm"
   Group "Group_11" at 1071,479 size 114x111
   Group "Group_15" at 1067,430 size 123x172
      HorizontalMovement <- "Station 2 Door Close"
   Group "Group_24" at 1002,13 size 65x83; PictureOff "Pushbutton_Emergency_Off_256c"; PictureOn "Pushbutton_Emergency_On_256c"
   SymbolLibrary "Symbol library_46" at 882,497 size 90x10
      Visibility <- "Station 2 Hide Vessel Tubing"
      Appearance <- "Station 2 Tubing Vessel"
   SymbolLibrary "Symbol library_25" at 870,479 size 10x20
      Appearance <- "Station 2 Tubing Vessel"
   SymbolLibrary "Symbol library_36" at 870,221 size 10x263
      Appearance <- "Station 2 Pump Tubing"
   Group "Group_19" at 857,187 size 38x40
   SymbolLibrary "Symbol library_44" at 875,253 size 159x73
   GraphicView "Graphic view_4" at 955,263 size 46x48; Picture "Graphic_1"
      Visibility <- "Station 2 Pump Rad Alarm"
   Group "Group_26" at 1070,33 size 153x83
   Group "Group_27" at 1070,34 size 153x132
   Group "Group_14" at 220,257 size 141x31; Text 'SYSTEM 1'
   Group "Group_25" at 654,278 size 141x31; Text 'SYSTEM 1'
   TextField "Text field_32" at 675,442 size 102x25; Text 'MATERIAL'
   TextField "Text field_33" at 689,459 size 66x25; Text 'VAULT'
   Group "Group_28" at 1085,257 size 141x31; Text 'SYSTEM 1'
   Button "Button_3" at 664,12 size 115x69; TextOff 'SILENCE BUZZER'
      Visibility <- "Estop Active"
      on Press: function_b14e0dd5("Buzzer Reset", 0)
   Group "Group_29" at 653,241 size 139x31; Text 'SYSTEM 1'
   IOField "I/O field_3" at 374,330 size 177x33; FormatPattern 999999; Unit  uRem/h
      ProcessValue <- "Station 1 Pump Rad Level"
   IOField "I/O field_12" at 371,628 size 181x33; FormatPattern 999999; Unit  uRem/h
      ProcessValue <- "Station 1 Vessel Rad Level"
   IOField "I/O field_14" at 633,150 size 178x33; FormatPattern 999999; Unit  uRem/h
      ProcessValue <- "Waste Rad Level"
   IOField "I/O field_23" at 882,330 size 179x33; FormatPattern 999999; Unit  uRem/h
      ProcessValue <- "Station 2 Pump Rad Level"
   IOField "I/O field_24" at 885,628 size 179x33; FormatPattern 999999; Unit  uRem/h
      ProcessValue <- "Station 2 Vessel Rad Level"
   Rectangle "Rectangle_2" at 252,480 size 112x111
      Visibility <- "Station 1 Door Lock Bypass"
   TextField "Text field_1" at 256,484 size 110x23; Text 'DOOR LOCK'
      Visibility <- "Station 1 Door Lock Bypass"
   Button "Button_2" at 267,510 size 80x70; TextOff 'BYPASS'
      on Press: function_b14e0dd5("Station 1 Door Lock Open", 0)
      Visibility <- "Station 1 Door Lock Bypass"
      ObjectEnable <- "Station 1 Process Running"
   GraphicIOField "PlotLight_Round_GN_2" at 321,512 size 22x23; PictureOn "PilotLight_Round_GN_On_256c"; PictureOff "PilotLight_Round_GN_Off_256c"
      ProcessValue <- "Station 1 Door Lock Open"
      Visibility <- "Station 1 Door Lock Bypass"
   Rectangle "Rectangle_3" at 220,135 size 170x31
      Visibility <- "Station 1 Manual Mode"
   TextField "Text field_2" at 224,135 size 163x27; Text 'MANUAL MODE'
      Visibility <- "Station 1 Manual Mode"
   TextField "Text field_12" at 226,35 size 173x39; Text 'STATION 1'
   Group "Group_5" at 448,519 size 24x41
   Group "Group_7" at 249,431 size 34x34
   Group "Group_8" at 331,431 size 34x34
   Group "Group_9" at 246,467 size 123x137
   Rectangle "Rectangle_21" at 246,467 size 123x137
      Visibility <- "Station 1 Door Locked"
   Rectangle "Rectangle_22" at 341,506 size 11x54
      Visibility <- "Station 1 Door Locked"
   Rectangle "Rectangle_23" at 485,36 size 153x79
      Visibility <- "Station 1 Auto Info"
   TextField "Text field_17" at 491,75 size 121x35; Text 'COMPLETED:'
      Visibility <- "Station 1 Auto Info"
   IOField "I/O field_4" at 595,82 size 27x22; FormatPattern 99
      ProcessValue <- "Station 1 Auto Current Rinse Num"
      Visibility <- "Station 1 Auto Info"
   IOField "I/O field_5" at 595,61 size 27x24; FormatPattern 99
      ProcessValue <- "Station 1 Auto Number of Rinses"
      Visibility <- "Station 1 Auto Info"
   TextField "Text field_18" at 534,60 size 62x25; Text 'TOTAL:'
      Visibility <- "Station 1 Auto Info"
   TextField "Text field_19" at 491,32 size 143x37; Text 'RINSE SEQUENCE'
      Visibility <- "Station 1 Auto Info"
   Rectangle "Rectangle_24" at 485,36 size 153x125
      Visibility <- "Station 1 Auto Info"
   TextField "Text field_23" at 497,130 size 121x35; Text 'COMPLETED:'
      Visibility <- "Station 1 Auto Info"
   IOField "I/O field_8" at 591,136 size 27x22; FormatPattern 99
      ProcessValue <- "Station 1 Auto Current Rinse Num"
      Visibility <- "Station 1 Auto Info"
   IOField "I/O field_9" at 591,97 size 27x24; FormatPattern 99
      ProcessValue <- "Station 1 Auto Number of Rinses"
      Visibility <- "Station 1 Auto Info"
   TextField "Text field_24" at 534,117 size 57x22; Text 'TOTAL:'
      Visibility <- "Station 1 Auto Info"
   TextField "Text field_25" at 498,73 size 126x37; Text 'RINSE SEQUENCE'
      Visibility <- "Station 1 Auto Info"
   TextField "Text field_26" at 500,33 size 130x37; Text 'RAD CONTROL'
      Visibility <- "Station 1 Auto Info"
   TextField "Text field_27" at 490,54 size 63x37; Text 'RAD SP:'
      Visibility <- "Station 1 Auto Info"
   TextField "Text field_28" at 535,98 size 50x22; Text 'FINAL:'
      Visibility <- "Station 1 Auto Info"
   IOField "I/O field_10" at 548,60 size 45x24; FormatPattern 9999
      ProcessValue <- "S1 Auto Rinse to RAD Level"
      Visibility <- "Station 1 Auto Info"
   TextField "Text field_29" at 590,54 size 48x37; Text 'Rad/h'
      Visibility <- "Station 1 Auto Info"
   IOField "I/O field_11" at 591,116 size 27x24; FormatPattern 99
      ProcessValue <- "Station 1 RAD Complete Rinses"
      Visibility <- "Station 1 Auto Info"
   SymbolLibrary "Symbol library_11" at 540,195 size 19x20
      Appearance <- "Station 1 Valve Rinse"
   SymbolLibrary "Symbol library_13" at 558,195 size 19x20
      Appearance <- "Station 1 Valve Drain"
   SymbolLibrary "Symbol library_14" at 549,205 size 19x20
      Appearance <- "Station 1 Valve Pump"
   TextField "Text field_4" at 432,217 size 65x29; Text 'STOP'
      Visibility <- "Station 1 Pump Run"
   TextField "Text field_5" at 412,217 size 55x29; Text 'RUN'
      Visibility <- "Station 1 Pump Run"
   TextField "Text field_6" at 464,217 size 58x29; Text 'FWD'
      Visibility <- "Station 1 PMP FWD"
   TextField "Text field_7" at 465,217 size 50x29; Text 'REV'
      Visibility <- "Station 1 PMP REV"
   Rectangle "Rectangle_30" at 808,134 size 170x31
      Visibility <- "Station 2 Manual Mode"
   TextField "Text field_35" at 812,134 size 163x27; Text 'MANUAL MODE'
      Visibility <- "Station 2 Manual Mode"
   TextField "Text field_45" at 814,34 size 173x39; Text 'STATION 2'
   TextField "Text field_37" at 938,218 size 65x29; Text 'STOP'
      Visibility <- "Station 2 Pump Run"
   TextField "Text field_38" at 918,218 size 55x29; Text 'RUN'
      Visibility <- "Station 2 Pump Run"
   TextField "Text field_39" at 970,218 size 58x29; Text 'FWD'
      Visibility <- "Station 2 PMP FWD"
   TextField "Text field_40" at 971,218 size 50x29; Text 'REV'
      Visibility <- "Station 2 PMP REV"
   Group "Group_20" at 959,518 size 24x41
   Rectangle "Rectangle_29" at 1071,479 size 112x111
      Visibility <- "Station 2 Door Lock Bypass"
   TextField "Text field_22" at 1075,483 size 110x23; Text 'DOOR LOCK'
      Visibility <- "Station 2 Door Lock Bypass"
   Button "Button_1" at 1086,509 size 80x70; TextOff 'BYPASS'
      on Press: function_b14e0dd5("Station 2 Door Lock Open", 0)
      Visibility <- "Station 2 Door Lock Bypass"
      ObjectEnable <- "Station 2 Process Running"
   GraphicIOField "PlotLight_Round_GN_1" at 1140,511 size 22x23; PictureOff "PilotLight_Round_GN_Off_256c"; PictureOn "PilotLight_Round_GN_On_256c"
      ProcessValue <- "Station 2 Door Lock Open"
      Visibility <- "Station 2 Door Lock Bypass"
   Group "Group_22" at 1070,430 size 34x34
   Group "Group_23" at 1152,430 size 34x34
   Rectangle "Rectangle_50" at 1067,465 size 123x137
      Visibility <- "Station 2 Door Locked"
   Rectangle "Rectangle_51" at 1084,505 size 11x54
      Visibility <- "Station 2 Door Locked"
   Switch "Pushbutton_Emergency_1" at 1004,35 size 60x61; CaptionText 'Switch'; TextOff '0'; TextOn '1'; PictureOff "Pushbutton_Emergency_Off_256c"; PictureOn "Pushbutton_Emergency_On_256c"
      Visibility <- "Station 2 Estop PB Active"
      ProcessValue <- "Station 2 Estop PB Active"
   TextField "Text field_53" at 1002,13 size 65x25; Text 'ESTOP'
      Visibility <- "Station 2 Estop PB Active"
   SymbolLibrary "Symbol library_40" at 876,197 size 19x20
      Appearance <- "Station 2 Valve Rinse"
   SymbolLibrary "Symbol library_41" at 857,197 size 19x20
      Appearance <- "Station 2 Valve Drain"
   SymbolLibrary "Symbol library_42" at 866,207 size 19x20
      Appearance <- "Station 2 Valve Pump"
   Rectangle "Rectangle_52" at 1070,37 size 153x79
      Visibility <- "Station 2 Auto Info"
   TextField "Text field_50" at 1076,76 size 121x35; Text 'COMPLETED:'
      Visibility <- "Station 2 Auto Info"
   IOField "I/O field_21" at 1180,83 size 27x22; FormatPattern 99
      ProcessValue <- "Station 2 Auto Current Rinse Num"
      Visibility <- "Station 2 Auto Info"
   IOField "I/O field_22" at 1180,62 size 27x24; FormatPattern 99
      ProcessValue <- "Station 2 Auto Number of Rinses"
      Visibility <- "Station 2 Auto Info"
   TextField "Text field_51" at 1119,61 size 62x25; Text 'TOTAL:'
      Visibility <- "Station 2 Auto Info"
   TextField "Text field_52" at 1075,33 size 146x37; Text 'RINSE SEQUENCE'
      Visibility <- "Station 2 Auto Info"
   Rectangle "Rectangle_53" at 1070,37 size 153x125
      Visibility <- "Station 2 Auto Info"
   TextField "Text field_55" at 1082,131 size 121x35; Text 'COMPLETED:'
      Visibility <- "Station 2 Auto Info"
   IOField "I/O field_25" at 1176,137 size 27x22; FormatPattern 99
      ProcessValue <- "Station 2 Auto Current Rinse Num"
      Visibility <- "Station 2 Auto Info"
   IOField "I/O field_26" at 1176,98 size 27x24; FormatPattern 99
      ProcessValue <- "Station 2 Auto Number of Rinses"
      Visibility <- "Station 2 Auto Info"
   TextField "Text field_56" at 1119,118 size 57x22; Text 'TOTAL:'
      Visibility <- "Station 2 Auto Info"
   TextField "Text field_57" at 1082,74 size 126x37; Text 'RINSE SEQUENCE'
      Visibility <- "Station 2 Auto Info"
   TextField "Text field_58" at 1085,34 size 130x37; Text 'RAD CONTROL'
      Visibility <- "Station 2 Auto Info"
   TextField "Text field_59" at 1075,55 size 63x37; Text 'RAD SP:'
      Visibility <- "Station 2 Auto Info"
   TextField "Text field_60" at 1120,99 size 50x22; Text 'FINAL:'
      Visibility <- "Station 2 Auto Info"
   IOField "I/O field_27" at 1133,61 size 45x24; FormatPattern 9999
      ProcessValue <- "S2 Auto Rinse to RAD Level"
      Visibility <- "Station 2 Auto Info"
   TextField "Text field_61" at 1175,55 size 48x37; Text 'Rad/h'
      Visibility <- "Station 2 Auto Info"
   IOField "I/O field_28" at 1176,117 size 27x24; FormatPattern 99
      ProcessValue <- "Station 2 RAD Complete Rinses"
      Visibility <- "Station 2 Auto Info"
   Rectangle "Rectangle_25" at 220,257 size 139x31
      Visibility <- "Station 1 Water Supply Interlock"
   TextField "Text field_30" at 223,257 size 138x29; Text 'INTERLOCK'
      Visibility <- "Station 1 Water Supply Interlock"
   Rectangle "Rectangle_32" at 654,278 size 139x31
      Visibility <- "Waste Drum Interlock"
   TextField "Text field_31" at 657,278 size 138x29; Text 'INTERLOCK'
      Visibility <- "Waste Drum Interlock"
   Rectangle "Rectangle_33" at 1085,257 size 139x31
      Visibility <- "Station 2 Water Supply Interlock"
   TextField "Text field_34" at 1088,257 size 138x29; Text 'INTERLOCK'
      Visibility <- "Station 2 Water Supply Interlock"
   Rectangle "Rectangle_54" at 653,241 size 139x31
      Visibility <- "UM Hi Level SW"
   TextField "Text field_47" at 656,241 size 123x29; Text 'HI LEVEL'
      Visibility <- "UM Hi Level SW"

screen "S2 Setup Screen" 1280x700, template "Navigation"
   TextField "Text field_3" at 197,62 size 258x34; Text 'AUTO MODE SETUP'
   Group "Group_1" at 198,6 size 466x49; Text 'SYSTEM 1'
   Group "Group_3" at 472,259 size 264x164; Text 'WASTE RAMP'; Authorization "Maintenance"
   Group "Group_4" at 472,422 size 265x164; Authorization "Maintenance"
   Group "Group_5" at 807,406 size 332x180; Authorization "Maintenance"; FormatPattern 99999
   Group "Group_6" at 808,201 size 448x185; Authorization "Maintenance"
   Group "Group" at 198,96 size 275x290; Authorization "Maintenance"
   Group "Group_2" at 198,385 size 275x227; Authorization "Maintenance"
   Group "Group_7" at 472,96 size 264x164; Authorization "Maintenance"
   TextField "Text field_15" at 209,6 size 455x43; Text 'STATION 2 SETUP SCREEN'
   TextField "Text field_12" at 237,101 size 206x29; Text 'PROCESS TIMERS'
   TextField "Text field_16" at 203,319 size 129x27; Text 'TOTAL NUM'
   IOField "I/O field_7" at 326,324 size 130x48; Authorization "Maintenance"; FormatPattern 999
      ProcessValue <- "S2 Auto Number of Rinses"
   TextField "Text field_17" at 203,280 size 124x27; Text 'TIME (ms):'
   IOField "I/O field_8" at 325,261 size 130x48; Authorization "Maintenance"; FormatPattern 99999
      ProcessValue <- "S2 Auto Rinse Run Time"
   TextField "Text field_18" at 202,258 size 72x27; Text 'RINSE'
   IOField "I/O field_9" at 324,199 size 130x48; Authorization "Maintenance"; FormatPattern 99999
      ProcessValue <- "S2 Auto Drain Run Time"
   TextField "Text field_19" at 203,196 size 75x27; Text 'DRAIN'
   TextField "Text field_20" at 204,218 size 124x27; Text 'TIME (ms):'
   TextField "Text field_21" at 203,342 size 93x27; Text 'CYCLES:'
   IOField "I/O field_15" at 324,137 size 130x48; Authorization "Maintenance"; FormatPattern 99999
      ProcessValue <- "S2 Auto Remove Run Time"
   TextField "Text field_34" at 203,134 size 94x27; Text 'REMOVE'
   TextField "Text field_35" at 204,156 size 124x27; Text 'TIME (ms):'
   TextField "Text field_4" at 235,389 size 210x29; Text 'PUMP MAX SPEED'
   TextField "Text field_5" at 221,491 size 83x27; Text 'DRAIN:'
   IOField "I/O field_1" at 304,483 size 101x48; Authorization "Maintenance"; FormatPattern 999
      ProcessValue <- "S2 Auto Pump Drain Max Speed"
   TextField "Text field_6" at 226,552 size 80x27; Text 'RINSE:'
   IOField "I/O field_2" at 305,545 size 101x48; Authorization "Maintenance"; FormatPattern 999
      ProcessValue <- "S2 Auto Pump Rinse Max Speed"
   TextField "Text field_13" at 409,552 size 51x27; Text 'RPM'
   TextField "Text field_14" at 407,491 size 51x27; Text 'RPM'
   TextField "Text field_36" at 204,429 size 102x27; Text 'REMOVE:'
   IOField "I/O field_17" at 304,421 size 101x48; Authorization "Maintenance"; FormatPattern 999
      ProcessValue <- "S2 Auto Pump Remove Max Speed"
   TextField "Text field_37" at 407,429 size 51x27; Text 'RPM'
   TextField "Text field_1" at 537,263 size 154x29; Text 'DRAIN RAMP'
   TextField "Text field_7" at 477,307 size 124x27; Text 'NO. STEPS:'
   IOField "I/O field_3" at 594,299 size 128x48; Authorization "Maintenance"; FormatPattern 999
      ProcessValue <- "S2 Auto Ramp Drain Step"
   TextField "Text field_8" at 476,368 size 124x27; Text 'TIME (ms):'
   IOField "I/O field_4" at 593,361 size 128x48; Authorization "Maintenance"; FormatPattern 99999
      ProcessValue <- "S2 Auto Ramp Drain Time"
   TextField "Text field_9" at 539,426 size 150x29; Text 'RINSE RAMP'
   TextField "Text field_10" at 478,472 size 124x27; Text 'NO. STEPS:'
   IOField "I/O field_5" at 598,462 size 125x48; Authorization "Maintenance"; FormatPattern 999
      ProcessValue <- "S2 Auto Ramp Rinse Step"
   TextField "Text field_11" at 477,531 size 124x27; Text 'TIME (ms):'
   IOField "I/O field_6" at 599,524 size 125x48; Authorization "Maintenance"; FormatPattern 99999
      ProcessValue <- "S2 Auto Ramp Rinse Time"
   TextField "Text field_2" at 858,411 size 232x29; Text 'PUMP PARAMETERS'
   TextField "Text field_22" at 812,531 size 154x27; Text 'VOLUME (ml):'
   IOField "I/O field_10" at 970,512 size 130x48; Authorization "Maintenance"; FormatPattern 99.999
      ProcessValue <- "S2 Pump Stroke Volume"
   TextField "Text field_23" at 811,509 size 155x27; Text 'PUMP STROKE'
   IOField "I/O field_11" at 969,450 size 130x48; Authorization "Maintenance"; FormatPattern 99.99
      ProcessValue <- "S2 Pump Factor"
   TextField "Text field_24" at 812,447 size 64x27; Text 'PUMP'
   TextField "Text field_25" at 813,469 size 97x27; Text 'FACTOR:'
   IOField "I/O field_12" at 1089,211 size 128x48; Authorization "Maintenance"; FormatPattern 999.99
      ProcessValue <- "Station 2 Container Water Supply Volume"
   IOField "I/O field_13" at 1089,268 size 128x48; Authorization "Maintenance"; FormatPattern 999
      ProcessValue <- "Station 2 Water Supply Alarm SP"
   TextField "Text field_26" at 816,222 size 286x29; Text 'WATER SUPPLY VOLUME'
   TextField "Text field_27" at 891,287 size 207x29; Text 'ALARM SETPOINT'
   TextField "Text field_28" at 890,266 size 183x29; Text 'WATER SUPPLY'
   TextField "Text field_29" at 1219,222 size 18x29; Text 'L'
   TextField "Text field_30" at 1219,277 size 31x29; Text '%'
   IOField "I/O field_14" at 1089,325 size 128x48; Authorization "Maintenance"; FormatPattern 999
      ProcessValue <- "Station 2 Water Supply Interlock SP"
   TextField "Text field_31" at 841,344 size 261x29; Text 'INTERLOCK SETPOINT'
   TextField "Text field_32" at 840,323 size 183x29; Text 'WATER SUPPLY'
   TextField "Text field_33" at 1219,334 size 31x29; Text '%'
   TextField "Text field_38" at 526,100 size 174x29; Text 'REMOVE RAMP'
   TextField "Text field_41" at 477,144 size 124x27; Text 'NO. STEPS:'
   IOField "I/O field_18" at 594,136 size 128x48; Authorization "Maintenance"; FormatPattern 999
      ProcessValue <- "S2 Auto Ramp Remove Step"
   TextField "Text field_42" at 476,205 size 124x27; Text 'TIME (ms):'
   IOField "I/O field_19" at 593,198 size 128x48; Authorization "Maintenance"; FormatPattern 99999
      ProcessValue <- "S2 Auto Ramp Remove Time"

screen "S1 Manual Mode" 1280x700, template "Navigation"
   on ClearScreen: SetBit("S1 Setup Data_Leave Manual Screen")
   on GenerateScreen: ResetBit("S1 Setup Data_Leave Manual Screen")
   Group "Group_3" at 492,12 size 427x42; Text 'SYSTEM 1'
   Group "Group_10" at 1142,98 size 112x111
   Switch "Pushbutton_Emergency" at 932,26 size 60x61; CaptionText 'Switch'; TextOff '0'; TextOn '1'; PictureOff "Pushbutton_Emergency_Off_256c"; PictureOn "Pushbutton_Emergency_On_256c"
      Visibility <- "Station 1 Estop PB Active"
      ProcessValue <- "Station 1 Estop PB Active"
   TextField "Text field_17" at 930,4 size 65x25; Text 'ESTOP'
      Visibility <- "Station 1 Estop PB Active"
   Rectangle "Rectangle_4" at 431,101 size 697x468
      Appearance <- "Station 1 Run State"
   SymbolLibrary "Symbol library_18" at 693,190 size 151x16
      Appearance <- "Station 1 Tubing Rinse"
   SymbolLibrary "Symbol library_13" at 855,223 size 15x255
      Appearance <- "Station 1 Pump Tubing"
   SymbolLibrary "Symbol library_2" at 568,235 size 298x124
   SymbolLibrary "Symbol library_21" at 890,190 size 93x14
      Appearance <- "Station 1 Tubing Drain"
   TextField "Text field_9" at 609,181 size 85x32; Text 'RINSE'
   TextField "Text field_10" at 980,163 size 151x32; Text 'UNWANTED'
   TextField "Text field_14" at 844,472 size 38x32; Text 'SV'
   Group "Group_4" at 648,369 size 156x40
   Group "Group_13" at 908,216 size 108x188; TextOff 'WASTE'
   Group "Group_11" at 991,444 size 114x111; Authorization "Maintenance"
   Group "Group_6" at 832,154 size 64x82
   Group "Group_17" at 194,13 size 215x125; Authorization "Maintenance"
   Group "Group_12" at 617,416 size 213x129; Text 'PUMP SPEED'
   Group "Group" at 452,418 size 144x122; TextOff 'OFF'
   Button "Button_13" at 487,456 size 74x63; TextOff 'SLEW'
      Visibility <- "Station 1 Manual Mode"
   Group "Group_14" at 1143,222 size 120x111; TextOff 'BYPASS'; Text 'DOOR LOCK'
   Group "Group_5" at 452,214 size 105x188
   Button "Button_9" at 465,251 size 74x63; TextOff 'FWD'
      Visibility <- "Station 1 Manual Mode"
   Button "Button_10" at 467,330 size 74x63; TextOff 'REV'
      Visibility <- "Station 1 Manual Mode"
   Group "Group_9" at 482,276 size 532x42; Text 'SYSTEM 1'
   TextField "Text field_18" at 981,186 size 135x32; Text 'MATERIAL'
   IOField "I/O field_2" at 648,93 size 159x56; FormatPattern 9999.9
      ProcessValue <- "Station 1 MM Feedback RPM"
   TextField "Text field_20" at 650,59 size 165x32; Text 'PUMP SPEED'
   Rectangle "Rectangle_16" at 650,96 size 154x49
      Visibility <- "Station 1 Manual Mode"
   TextField "Text field_21" at 697,148 size 61x32; Text 'RPM'
   Group "Group_8" at 619,274 size 194x44
   Group "Group_15" at 619,274 size 194x44
   Group "Group_16" at 562,579 size 419x95
   Group "Group_18" at 562,580 size 419x93
   TextField "Text field_13" at 502,12 size 417x39; Text 'STATION 1 MANUAL MODE'
   Rectangle "Rectangle_11" at 482,276 size 518x42
      Visibility <- "Station 1 Process Running"
   TextField "Text field_16" at 494,276 size 520x39; Text 'STATION 1 IN AUTOMATIC MODE'
      Visibility <- "Station 1 Process Running"
   Rectangle "Rectangle_13" at 1142,98 size 112x111
      Visibility <- "CurrentGroupNum"
   TextField "Text field_15" at 1151,102 size 97x23; Text 'RAD LOCK'
      Visibility <- "CurrentGroupNum"
   Button "Button_15" at 1157,128 size 80x70; TextOff 'BYPASS'; Authorization "Health_Physics"
      on Press: InvertBit("Station 1 Rad Lock Bypass")
      Visibility <- "CurrentGroupNum"
   GraphicIOField "PlotLight_Round_GN_6" at 1211,130 size 22x23; PictureOn "PilotLight_Round_GN_On_256c"; PictureOff "PilotLight_Round_GN_Off_256c"
      Visibility <- "CurrentGroupNum"
      ProcessValue <- "Station 1 Rad Lock Bypass"
   TextField "Text field_4" at 690,372 size 71x32; Text 'STOP'
      Visibility <- "Station 1 MM PMP Run"
   TextField "Text field_8" at 671,372 size 60x32; Text 'RUN'
      Visibility <- "Station 1 MM PMP Run"
   TextField "Text field_11" at 727,372 size 62x32; Text 'FWD'
      Visibility <- "Station 1 MM PMP FWD"
   TextField "Text field_12" at 730,372 size 55x32; Text 'REV'
      Visibility <- "Station 1 MM PMP REV"
   Group "Group_2" at 908,216 size 108x188; TextOff 'WASTE'
   Button "Button_11" at 922,253 size 74x63; TextOff 'UM'
      Visibility <- "Station 1 Manual Mode"
   Button "Button_12" at 922,331 size 74x63; TextOff 'RINSE'
      Visibility <- "Station 1 Manual Mode"
   TextField "Text field_6" at 916,218 size 85x32; Text 'VALVE'
   Button "Button_7" at 922,253 size 74x63; TextOff 'UM'
      on Press: ResetBit("Station 1 MM Valve Direction SW")
   Button "Button_8" at 922,331 size 74x63; TextOff 'RINSE'
      on Press: SetBit("Station 1 MM Valve Direction SW")
   GraphicIOField "PlotLight_Round_GN_3" at 974,331 size 22x23; PictureOn "PilotLight_Round_GN_On_256c"; PictureOff "PilotLight_Round_GN_Off_256c"
      ProcessValue <- "Station 1 MM Valve Direction SW"
   GraphicIOField "PlotLight_Round_GN_4" at 972,253 size 22x23; PictureOff "PilotLight_Round_GN_On_256c"; PictureOn "PilotLight_Round_GN_Off_256c"
      ProcessValue <- "Station 1 MM Valve Direction SW"
   TextField "Text field_2" at 456,422 size 140x32; Text 'PUMP RUN'
   Button "Button_4" at 487,456 size 74x63; TextOff 'SLEW'
      on Press: SetBit("Station 1 MM Pump Slew PB")
   GraphicIOField "PlotLight_Round_GN_1" at 536,458 size 22x23; PictureOn "PilotLight_Round_GN_On_256c"; PictureOff "PilotLight_Round_GN_Off_256c"
      ProcessValue <- "Station 1 MM Pump Slew PB"
   TextField "Text field_3" at 464,217 size 77x32; Text 'PUMP'
   Button "Button_5" at 465,251 size 74x63; TextOff 'FWD'
      on Press: SetBit("Station 1 MM Pump Dir FWD"); ResetBit("Station 1 MM Pump Dir REV")
   Button "Button_6" at 467,330 size 74x63; TextOff 'REV'
      on Press: SetBit("Station 1 MM Pump Dir REV"); ResetBit("Station 1 MM Pump Dir FWD")
   GraphicIOField "PlotLight_Round_GN_2" at 517,332 size 22x23; PictureOff "PilotLight_Round_GN_Off_256c"; PictureOn "PilotLight_Round_GN_On_256c"
      ProcessValue <- "Station 1 MM Pump Dir REV"
   GraphicIOField "PlotLight_Round_GN_5" at 516,253 size 22x23; PictureOn "PilotLight_Round_GN_On_256c"; PictureOff "PilotLight_Round_GN_Off_256c"
      ProcessValue <- "Station 1 MM Pump Dir FWD"
   Group "Group_1" at 617,416 size 213x129; Text 'PUMP SPEED'; FormatPattern 99999
   Rectangle "Rectangle_12" at 642,457 size 154x49
      Visibility <- "Station 1 Manual Mode"
   IOField "I/O field_1" at 639,454 size 159x56; FormatPattern 9999.9
      ProcessValue <- "Station 1 Pump Speed SP RPM"
   TextField "Text field_5" at 625,420 size 205x32; Text 'PUMP SPEED SP'
   TextField "Text field_7" at 685,510 size 61x32; Text 'RPM'
   TextField "Text field_22" at 995,448 size 110x23; Text 'DOOR LOCK'
   Button "Button_16" at 1006,474 size 80x70; TextOff 'BYPASS'; Authorization "Maintenance"
      on Press: function_b14e0dd5("Station 1 Door Lock Open", 0)
   GraphicIOField "PlotLight_Round_GN_7" at 1060,476 size 22x23; PictureOn "PilotLight_Round_GN_On_256c"; PictureOff "PilotLight_Round_GN_Off_256c"; Authorization "Maintenance"
      ProcessValue <- "Station 1 Door Lock Open"
   SymbolLibrary "Symbol library_4" at 832,180 size 32x36
      Appearance <- "Station 1 Valve Rinse"
   SymbolLibrary "Symbol library_3" at 864,180 size 32x36
      Appearance <- "Station 1 Valve Drain"
   SymbolLibrary "Symbol library_5" at 847,200 size 32x36
      Appearance <- "Station 1 Valve Pump"
   TextField "Text field_1" at 210,18 size 194x32; Text 'MANUAL MODE'
   Button "Button_2" at 310,57 size 74x63; TextOff 'OFF'; Authorization "Maintenance"
      on Press: ResetBit("Station 1 Manual Mode"); SetTag("Station 1 Pump Speed SP RPM", 0); ResetBit("Station 1 MM Pump Dir FWD"); ResetBit("Station 1 MM Valve Direction SW"); ResetBit("Station 1 MM Pump Dir REV"); ResetBit("Station 1 Warning 1"); ResetBit("Station 1 Warning 2")
   Group "Group_7" at 216,57 size 74x63; Authorization "Maintenance"
   Button "Button_1" at 216,57 size 74x63; TextOff 'ON'; Authorization "Maintenance"
      on Press: SetBit("Station 1 Manual Mode")
      ObjectEnable <- "Station 1 Process Running"
   GraphicIOField "PlotLight_Round_GN" at 268,61 size 22x23; PictureOn "PilotLight_Round_GN_On_256c"; PictureOff "PilotLight_Round_GN_Off_256c"; Authorization "Maintenance"
      ProcessValue <- "Station 1 Manual Mode"
   TextField "Text field_19" at 1144,226 size 119x21; Text 'RESET MOTOR'
   Button "Button_18" at 1160,252 size 80x70; TextOff 'RESET'
      on Press: InvertBit("Pump 1 Motor_Reset")
   GraphicIOField "PlotLight_Round_GN_9" at 1216,254 size 22x23; PictureOff "PilotLight_Round_GN_Off_256c"; PictureOn "PilotLight_Round_GN_On_256c"
      ProcessValue <- "Pump 1 Motor_Reset"
   TextField "Text field_26" at 562,637 size 419x37; Text 'Material may be radioactive!'
      Visibility <- "Station 1 Warning 1"
   TextField "Text field_25" at 606,607 size 279x37; Text 'from UM to the SV.'
      Visibility <- "Station 1 Warning 1"
   TextField "Text field_24" at 588,579 size 354x37; Text 'Material will be pumped'
      Visibility <- "Station 1 Warning 1"
   Rectangle "Rectangle_14" at 619,276 size 194x42
      Visibility <- "Station 1 Warning 1"
   TextField "Text field_23" at 634,274 size 164x43; Text 'CAUTION'
      Visibility <- "Station 1 Warning 1"
   Rectangle "Rectangle_17" at 619,276 size 194x42
      Visibility <- "Station 1 Warning 2"
   TextField "Text field_27" at 634,274 size 164x43; Text 'CAUTION'
      Visibility <- "Station 1 Warning 2"
   TextField "Text field_28" at 589,580 size 354x37; Text 'Material will be pumped'
      Visibility <- "Station 1 Warning 2"
   TextField "Text field_29" at 632,608 size 257x37; Text 'from SV to Rinse.'
      Visibility <- "Station 1 Warning 2"
   TextField "Text field_30" at 562,636 size 419x37; Text 'Material may be radioactive!'
      Visibility <- "Station 1 Warning 2"

screen "S1 Setup Screen" 1280x700, template "Navigation"
   TextField "Text field_3" at 218,61 size 258x34; Text 'AUTO MODE SETUP'
   Group "Group_1" at 222,7 size 466x49; Text 'SYSTEM 1'
   Group "Group_5" at 819,514 size 332x180; Authorization "Maintenance"; FormatPattern 99999
   Group "Group_6" at 818,133 size 448x186; Authorization "Maintenance"
   Group "Group" at 218,96 size 275x295; Authorization "Maintenance"
   Group "Group_8" at 818,324 size 447x186; Authorization "Maintenance"
   Group "Group_2" at 218,390 size 275x235; Authorization "Maintenance"
   Group "Group_7" at 492,96 size 275x164; Authorization "Maintenance"
   Group "Group_3" at 492,259 size 275x164; Authorization "Maintenance"
   Group "Group_4" at 492,422 size 275x164; Authorization "Maintenance"
   TextField "Text field_15" at 233,7 size 455x43; Text 'STATION 1 SETUP SCREEN'
   TextField "Text field_12" at 249,101 size 206x29; Text 'PROCESS TIMERS'
   TextField "Text field_16" at 223,319 size 129x27; Text 'TOTAL NUM'
   IOField "I/O field_7" at 346,324 size 130x48; Authorization "Maintenance"; FormatPattern 999
      ProcessValue <- "S1 Auto Number of Rinses"
   TextField "Text field_17" at 223,280 size 124x27; Text 'TIME (ms):'
   IOField "I/O field_8" at 345,261 size 130x48; Authorization "Maintenance"; FormatPattern 99999
      ProcessValue <- "S1 Auto Rinse Run Time"
   TextField "Text field_18" at 222,258 size 72x27; Text 'RINSE'
   IOField "I/O field_9" at 344,199 size 130x48; Authorization "Maintenance"; FormatPattern 99999
      ProcessValue <- "S1 Auto Drain Run Time"
   TextField "Text field_19" at 223,196 size 75x27; Text 'DRAIN'
   TextField "Text field_20" at 224,218 size 124x27; Text 'TIME (ms):'
   TextField "Text field_21" at 223,342 size 93x27; Text 'CYCLES:'
   IOField "I/O field_18" at 344,138 size 130x48; Authorization "Maintenance"; FormatPattern 99999
      ProcessValue <- "S1 Auto Remove Run Time"
   TextField "Text field_41" at 223,135 size 94x27; Text 'REMOVE'
   TextField "Text field_42" at 224,157 size 124x27; Text 'TIME (ms):'
   TextField "Text field_1" at 555,263 size 154x29; Text 'DRAIN RAMP'
   TextField "Text field_7" at 505,307 size 124x27; Text 'NO. STEPS:'
   IOField "I/O field_3" at 622,299 size 128x48; Authorization "Maintenance"; FormatPattern 999
      ProcessValue <- "S1 Auto Ramp Drain Step"
   TextField "Text field_8" at 504,368 size 124x27; Text 'TIME (ms):'
   IOField "I/O field_4" at 621,361 size 128x48; Authorization "Maintenance"; FormatPattern 99999
      ProcessValue <- "S1 Auto Ramp Drain Time"
   TextField "Text field_9" at 559,426 size 150x29; Text 'RINSE RAMP'
   TextField "Text field_10" at 503,472 size 124x27; Text 'NO. STEPS:'
   IOField "I/O field_5" at 623,462 size 125x48; Authorization "Maintenance"; FormatPattern 999
      ProcessValue <- "S1 Auto Ramp Rinse Step"
   TextField "Text field_11" at 502,531 size 124x27; Text 'TIME (ms):'
   IOField "I/O field_6" at 624,524 size 125x48; Authorization "Maintenance"; FormatPattern 99999
      ProcessValue <- "S1 Auto Ramp Rinse Time"
   TextField "Text field_4" at 251,394 size 210x29; Text 'PUMP MAX SPEED'
   TextField "Text field_5" at 247,503 size 83x27; Text 'DRAIN:'
   IOField "I/O field_1" at 325,495 size 101x48; Authorization "Maintenance"; FormatPattern 999
      ProcessValue <- "S1 Auto Pump Drain Max Speed"
   TextField "Text field_6" at 248,568 size 80x27; Text 'RINSE:'
   IOField "I/O field_2" at 325,559 size 101x48; Authorization "Maintenance"; FormatPattern 999
      ProcessValue <- "S1 Auto Pump Rinse Max Speed"
   TextField "Text field_13" at 424,568 size 51x27; Text 'RPM'
   TextField "Text field_14" at 425,503 size 51x27; Text 'RPM'
   TextField "Text field_37" at 230,440 size 102x27; Text 'REMOVE:'
   IOField "I/O field_17" at 324,432 size 101x48; Authorization "Maintenance"; FormatPattern 999
      ProcessValue <- "S1 Auto Pump Remove Max Speed"
   TextField "Text field_38" at 424,440 size 51x27; Text 'RPM'
   TextField "Text field_2" at 870,519 size 232x29; Text 'PUMP PARAMETERS'
   TextField "Text field_22" at 824,639 size 154x27; Text 'VOLUME (ml):'
   IOField "I/O field_10" at 982,620 size 130x48; Authorization "Maintenance"; FormatPattern 99.999
      ProcessValue <- "S1 Pump Stroke Volume"
   TextField "Text field_23" at 823,617 size 155x27; Text 'PUMP STROKE'
   IOField "I/O field_11" at 981,558 size 130x48; Authorization "Maintenance"; FormatPattern 99.99
      ProcessValue <- "S1 Pump Factor"
   TextField "Text field_24" at 824,555 size 64x27; Text 'PUMP'
   TextField "Text field_25" at 825,577 size 97x27; Text 'FACTOR:'
   IOField "I/O field_12" at 1099,143 size 128x48; Authorization "Maintenance"; FormatPattern 999.99
      ProcessValue <- "Station 1 Container Water Supply Volume"
   IOField "I/O field_13" at 1099,200 size 128x48; Authorization "Maintenance"; FormatPattern 999
      ProcessValue <- "Station 1 Water Supply Alarm SP"
   TextField "Text field_26" at 826,154 size 286x29; Text 'WATER SUPPLY VOLUME'
   TextField "Text field_27" at 901,219 size 207x29; Text 'ALARM SETPOINT'
   TextField "Text field_28" at 899,198 size 183x29; Text 'WATER SUPPLY'
   TextField "Text field_29" at 1229,154 size 18x29; Text 'L'
   TextField "Text field_30" at 1229,209 size 31x29; Text '%'
   IOField "I/O field_14" at 1099,259 size 128x48; Authorization "Maintenance"; FormatPattern 999
      ProcessValue <- "Station 1 Water Supply Interlock SP"
   TextField "Text field_31" at 851,278 size 261x29; Text 'INTERLOCK SETPOINT'
   TextField "Text field_32" at 850,257 size 183x29; Text 'WATER SUPPLY'
   TextField "Text field_33" at 1229,268 size 31x29; Text '%'
   IOField "I/O field_20" at 1099,334 size 131x48; Authorization "Maintenance"; FormatPattern 999.99
      ProcessValue <- "Waste Drum Volume"
   IOField "I/O field_21" at 1099,391 size 131x48; Authorization "Maintenance"; FormatPattern 999
      ProcessValue <- "Waste Drum Alarm SP"
   TextField "Text field_44" at 882,344 size 222x29; Text 'UM DRUM VOLUME'
   TextField "Text field_45" at 898,410 size 207x29; Text 'ALARM SETPOINT'
   TextField "Text field_46" at 844,389 size 264x29; Text 'UNWANTED MATERIAL'
   TextField "Text field_47" at 1231,345 size 18x29; Text 'L'
   TextField "Text field_48" at 1231,400 size 31x29; Text '%'
   IOField "I/O field_15" at 1099,448 size 131x48; Authorization "Maintenance"; FormatPattern 999
      ProcessValue <- "Waste Drum Level Interlock"
   TextField "Text field_34" at 849,467 size 261x29; Text 'INTERLOCK SETPOINT'
   TextField "Text field_35" at 844,446 size 264x29; Text 'UNWANTED MATERIAL'
   TextField "Text field_36" at 1231,457 size 31x29; Text '%'
   TextField "Text field_43" at 544,100 size 174x29; Text 'REMOVE RAMP'
   TextField "Text field_49" at 506,144 size 124x27; Text 'NO. STEPS:'
   IOField "I/O field_19" at 623,136 size 128x48; Authorization "Maintenance"; FormatPattern 999
      ProcessValue <- "S1Auto Ramp Remove Step"
   TextField "Text field_50" at 505,205 size 124x27; Text 'TIME (ms):'
   IOField "I/O field_22" at 622,198 size 128x48; Authorization "Maintenance"; FormatPattern 99999
      ProcessValue <- "S1Auto Ramp Remove Time"

